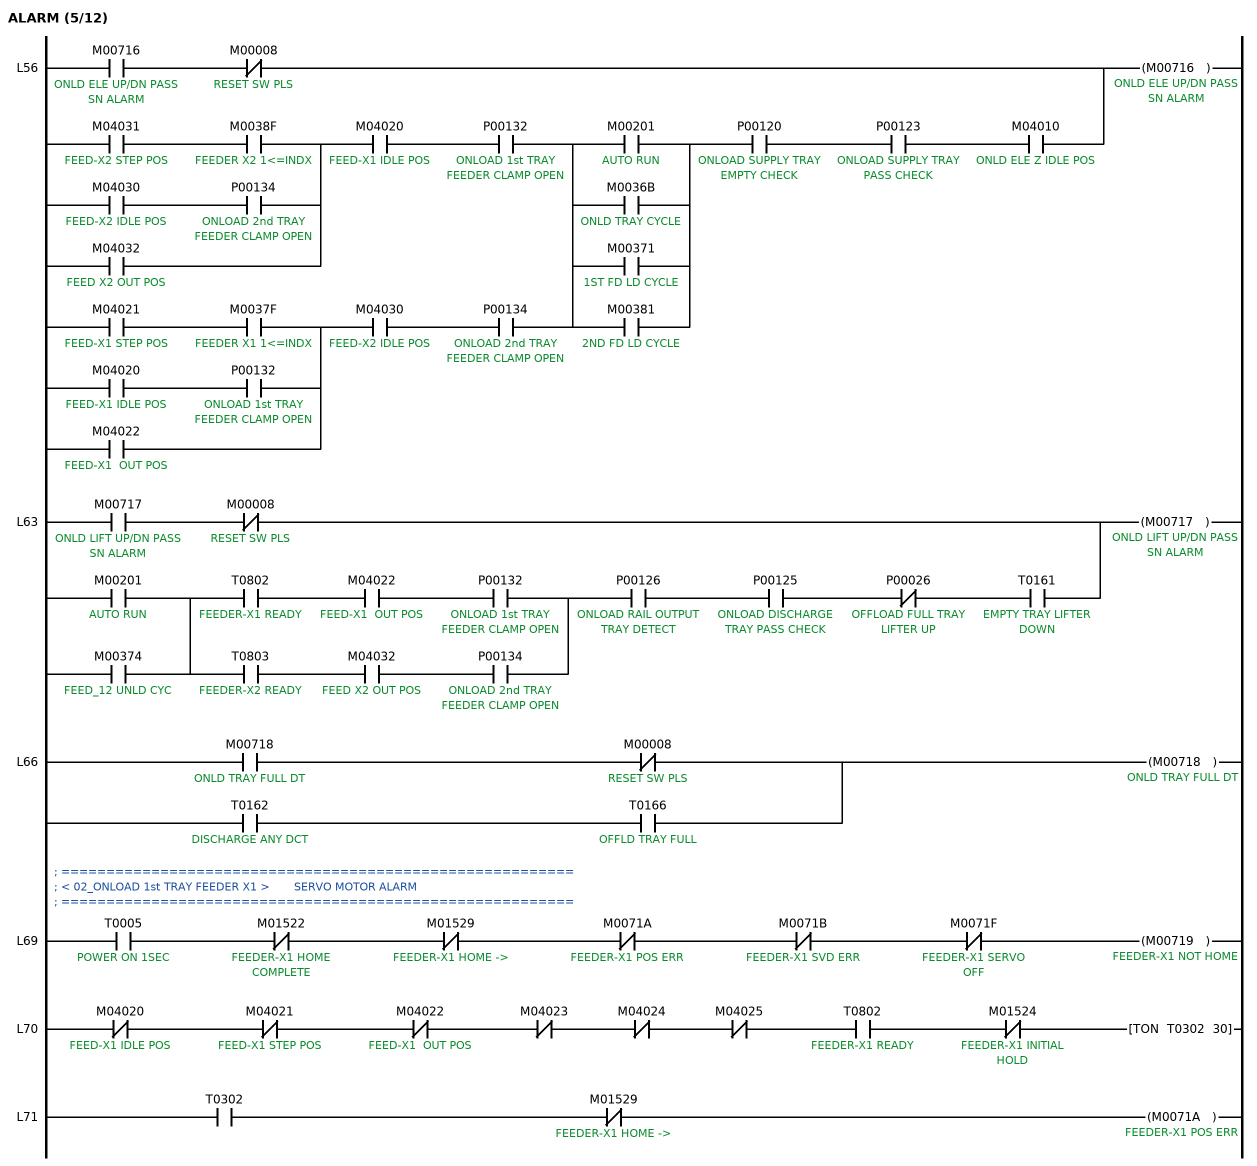
; L56
LOAD      M00716	// ONLD ELE UP/DN PASS SN ALARM
AND NOT   M00008	// RESET SW PLS
LOAD      M04031	// FEED-X2 STEP POS
AND       M0038F	// FEEDER X2 1<=INDX
LOAD      M04030	// FEED-X2 IDLE POS
AND       P00134	// ONLOAD 2nd TRAY FEEDER CLAMP OPEN
OR LOAD
OR        M04032	// FEED X2 OUT POS
AND       M04020	// FEED-X1 IDLE POS
AND       P00132	// ONLOAD 1st TRAY FEEDER CLAMP OPEN
LOAD      M04021	// FEED-X1 STEP POS
AND       M0037F	// FEEDER X1 1<=INDX
LOAD      M04020	// FEED-X1 IDLE POS
AND       P00132	// ONLOAD 1st TRAY FEEDER CLAMP OPEN
OR LOAD
OR        M04022	// FEED-X1  OUT POS
AND       M04030	// FEED-X2 IDLE POS
AND       P00134	// ONLOAD 2nd TRAY FEEDER CLAMP OPEN
OR LOAD
LOAD      M00201	// AUTO RUN
OR        M0036B	// ONLD TRAY CYCLE
OR        M00371	// 1ST FD LD CYCLE
OR        M00381	// 2ND FD LD CYCLE
AND LOAD
AND       P00120	// ONLOAD SUPPLY TRAY EMPTY CHECK
AND       P00123	// ONLOAD SUPPLY TRAY PASS CHECK
AND       M04010	// ONLD ELE Z IDLE POS
OR LOAD
OUT       M00716	// ONLD ELE UP/DN PASS SN ALARM
; L63
LOAD      M00717	// ONLD LIFT UP/DN PASS SN ALARM
AND NOT   M00008	// RESET SW PLS
LOAD      M00201	// AUTO RUN
OR        M00374	// FEED_12 UNLD CYC
LOAD      T0802	// FEEDER-X1 READY
AND       M04022	// FEED-X1  OUT POS
AND       P00132	// ONLOAD 1st TRAY FEEDER CLAMP OPEN
LOAD      T0803	// FEEDER-X2 READY
AND       M04032	// FEED X2 OUT POS
AND       P00134	// ONLOAD 2nd TRAY FEEDER CLAMP OPEN
OR LOAD
AND LOAD
AND       P00126	// ONLOAD RAIL OUTPUT TRAY DETECT
AND       P00125	// ONLOAD DISCHARGE TRAY PASS CHECK
AND NOT   P00026	// OFFLOAD FULL TRAY LIFTER UP
AND       T0161	// EMPTY TRAY LIFTER DOWN
OR LOAD
OUT       M00717	// ONLD LIFT UP/DN PASS SN ALARM
; L66
LOAD      M00718	// ONLD TRAY FULL DT
AND NOT   M00008	// RESET SW PLS
LOAD      T0162	// DISCHARGE ANY DCT
AND       T0166	// OFFLD TRAY FULL
OR LOAD
OUT       M00718	// ONLD TRAY FULL DT
// =========================================================
// 
//        < 02_ONLOAD 1st TRAY FEEDER X1 >       SERVO MOTOR ALARM
// 
// =========================================================
; L69
LOAD      T0005	// POWER ON 1SEC
AND NOT   M01522	// FEEDER-X1 HOME COMPLETE
AND NOT   M01529	// FEEDER-X1 HOME ->
AND NOT   M0071A	// FEEDER-X1 POS ERR
AND NOT   M0071B	// FEEDER-X1 SVD ERR
AND NOT   M0071F	// FEEDER-X1 SERVO OFF
OUT       M00719	// FEEDER-X1 NOT HOME
; L70
LOAD NOT  M04020	// FEED-X1 IDLE POS
AND NOT   M04021	// FEED-X1 STEP POS
AND NOT   M04022	// FEED-X1  OUT POS
AND NOT   M04023
AND NOT   M04024
AND NOT   M04025
AND       T0802	// FEEDER-X1 READY
AND NOT   M01524	// FEEDER-X1 INITIAL HOLD
TON       T0302 30
; L71
LOAD      T0302
AND NOT   M01529	// FEEDER-X1 HOME ->
OUT       M0071A	// FEEDER-X1 POS ERR

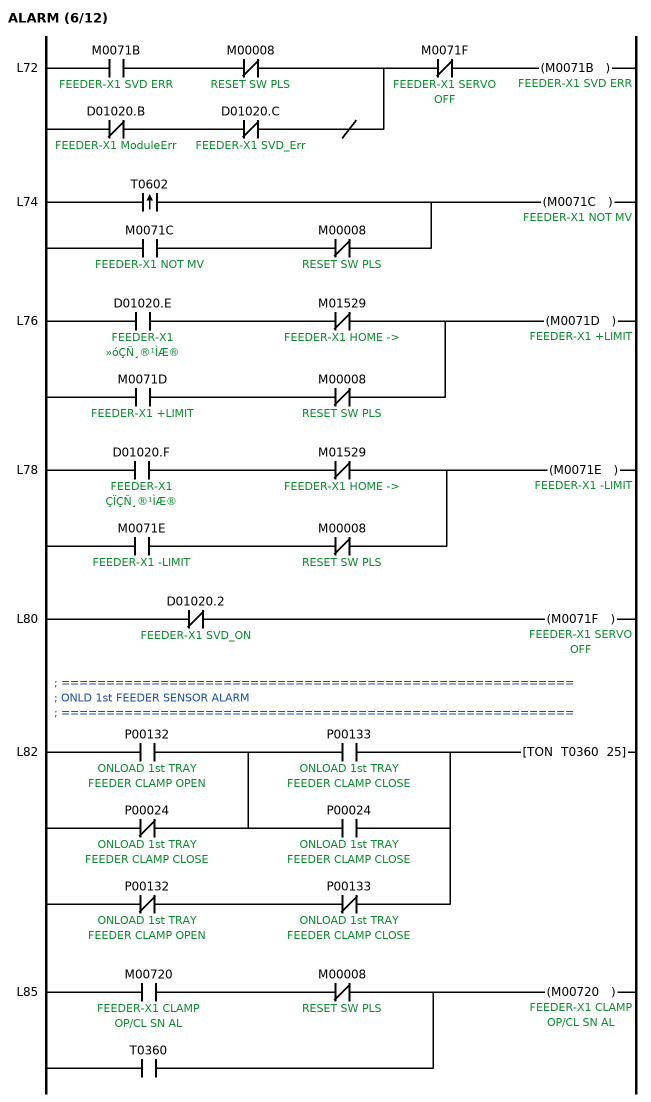
; L72
LOAD      M0071B	// FEEDER-X1 SVD ERR
AND NOT   M00008	// RESET SW PLS
LOAD NOT  D01020.B	// FEEDER-X1 ModuleErr
AND NOT   D01020.C	// FEEDER-X1 SVD_Err
NOT
OR LOAD
AND NOT   M0071F	// FEEDER-X1 SERVO OFF
OUT       M0071B	// FEEDER-X1 SVD ERR
; L74
LOADP     T0602
LOAD      M0071C	// FEEDER-X1 NOT MV
AND NOT   M00008	// RESET SW PLS
OR LOAD
OUT       M0071C	// FEEDER-X1 NOT MV
; L76
LOAD      D01020.E	// FEEDER-X1 »óÇÑ¸®¹ÌÆ®
AND NOT   M01529	// FEEDER-X1 HOME ->
LOAD      M0071D	// FEEDER-X1 +LIMIT
AND NOT   M00008	// RESET SW PLS
OR LOAD
OUT       M0071D	// FEEDER-X1 +LIMIT
; L78
LOAD      D01020.F	// FEEDER-X1 ÇÏÇÑ¸®¹ÌÆ®
AND NOT   M01529	// FEEDER-X1 HOME ->
LOAD      M0071E	// FEEDER-X1 -LIMIT
AND NOT   M00008	// RESET SW PLS
OR LOAD
OUT       M0071E	// FEEDER-X1 -LIMIT
; L80
LOAD NOT  D01020.2	// FEEDER-X1 SVD_ON
OUT       M0071F	// FEEDER-X1 SERVO OFF
// =========================================================
// 
//        ONLD 1st FEEDER SENSOR ALARM
// 
// =========================================================
; L82
LOAD      P00132	// ONLOAD 1st TRAY FEEDER CLAMP OPEN
OR NOT    P00024	// ONLOAD 1st TRAY FEEDER CLAMP CLOSE
LOAD      P00133	// ONLOAD 1st TRAY FEEDER CLAMP CLOSE
OR        P00024	// ONLOAD 1st TRAY FEEDER CLAMP CLOSE
AND LOAD
LOAD NOT  P00132	// ONLOAD 1st TRAY FEEDER CLAMP OPEN
AND NOT   P00133	// ONLOAD 1st TRAY FEEDER CLAMP CLOSE
OR LOAD
TON       T0360 25
; L85
LOAD      M00720	// FEEDER-X1 CLAMP OP/CL SN AL
AND NOT   M00008	// RESET SW PLS
OR        T0360
OUT       M00720	// FEEDER-X1 CLAMP OP/CL SN AL

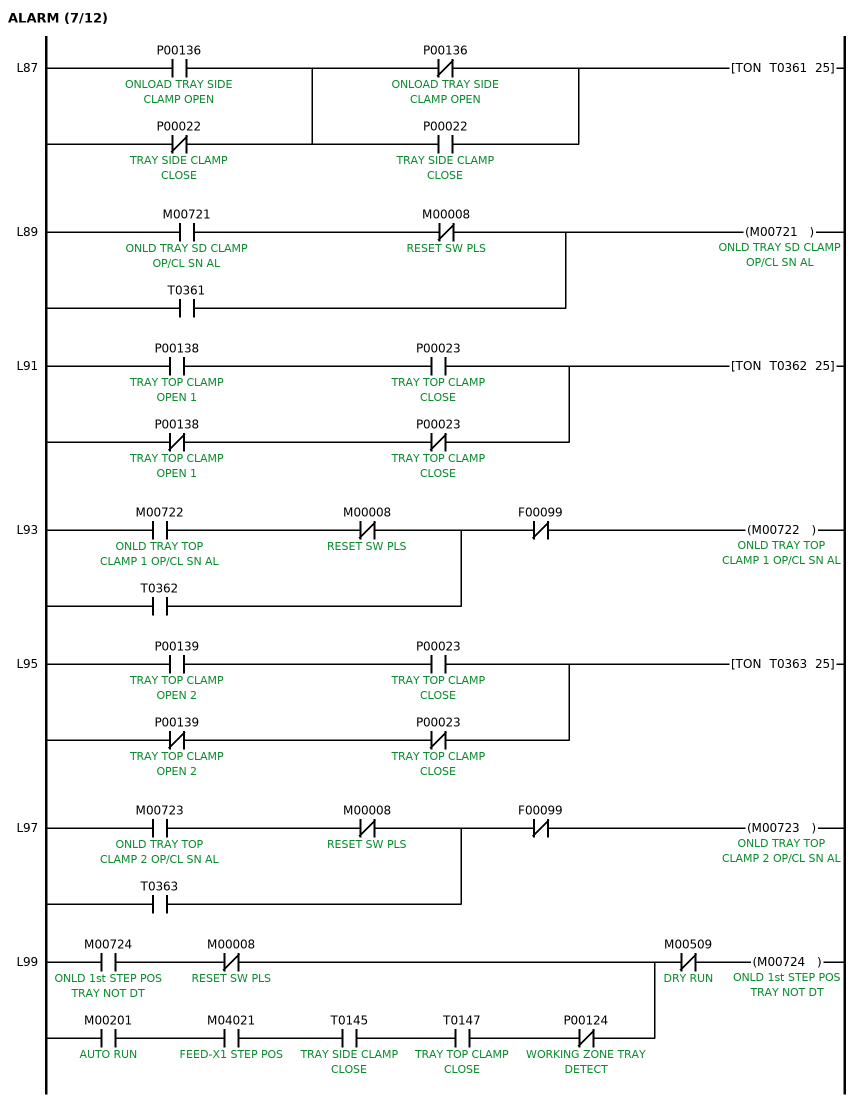
; L87
LOAD      P00136	// ONLOAD TRAY SIDE CLAMP OPEN
OR NOT    P00022	// TRAY SIDE CLAMP CLOSE
LOAD NOT  P00136	// ONLOAD TRAY SIDE CLAMP OPEN
OR        P00022	// TRAY SIDE CLAMP CLOSE
AND LOAD
TON       T0361 25
; L89
LOAD      M00721	// ONLD TRAY SD CLAMP OP/CL SN AL
AND NOT   M00008	// RESET SW PLS
OR        T0361
OUT       M00721	// ONLD TRAY SD CLAMP OP/CL SN AL
; L91
LOAD      P00138	// TRAY TOP CLAMP OPEN 1
AND       P00023	// TRAY TOP CLAMP CLOSE
LOAD NOT  P00138	// TRAY TOP CLAMP OPEN 1
AND NOT   P00023	// TRAY TOP CLAMP CLOSE
OR LOAD
TON       T0362 25
; L93
LOAD      M00722	// ONLD TRAY TOP CLAMP 1 OP/CL SN AL
AND NOT   M00008	// RESET SW PLS
OR        T0362
AND NOT   F00099
OUT       M00722	// ONLD TRAY TOP CLAMP 1 OP/CL SN AL
; L95
LOAD      P00139	// TRAY TOP CLAMP OPEN 2
AND       P00023	// TRAY TOP CLAMP CLOSE
LOAD NOT  P00139	// TRAY TOP CLAMP OPEN 2
AND NOT   P00023	// TRAY TOP CLAMP CLOSE
OR LOAD
TON       T0363 25
; L97
LOAD      M00723	// ONLD TRAY TOP CLAMP 2 OP/CL SN AL
AND NOT   M00008	// RESET SW PLS
OR        T0363
AND NOT   F00099
OUT       M00723	// ONLD TRAY TOP CLAMP 2 OP/CL SN AL
; L99
LOAD      M00724	// ONLD 1st STEP POS TRAY NOT DT
AND NOT   M00008	// RESET SW PLS
LOAD      M00201	// AUTO RUN
AND       M04021	// FEED-X1 STEP POS
AND       T0145	// TRAY SIDE CLAMP CLOSE
AND       T0147	// TRAY TOP CLAMP CLOSE
AND NOT   P00124	// WORKING ZONE TRAY DETECT
OR LOAD
AND NOT   M00509	// DRY RUN
OUT       M00724	// ONLD 1st STEP POS TRAY NOT DT

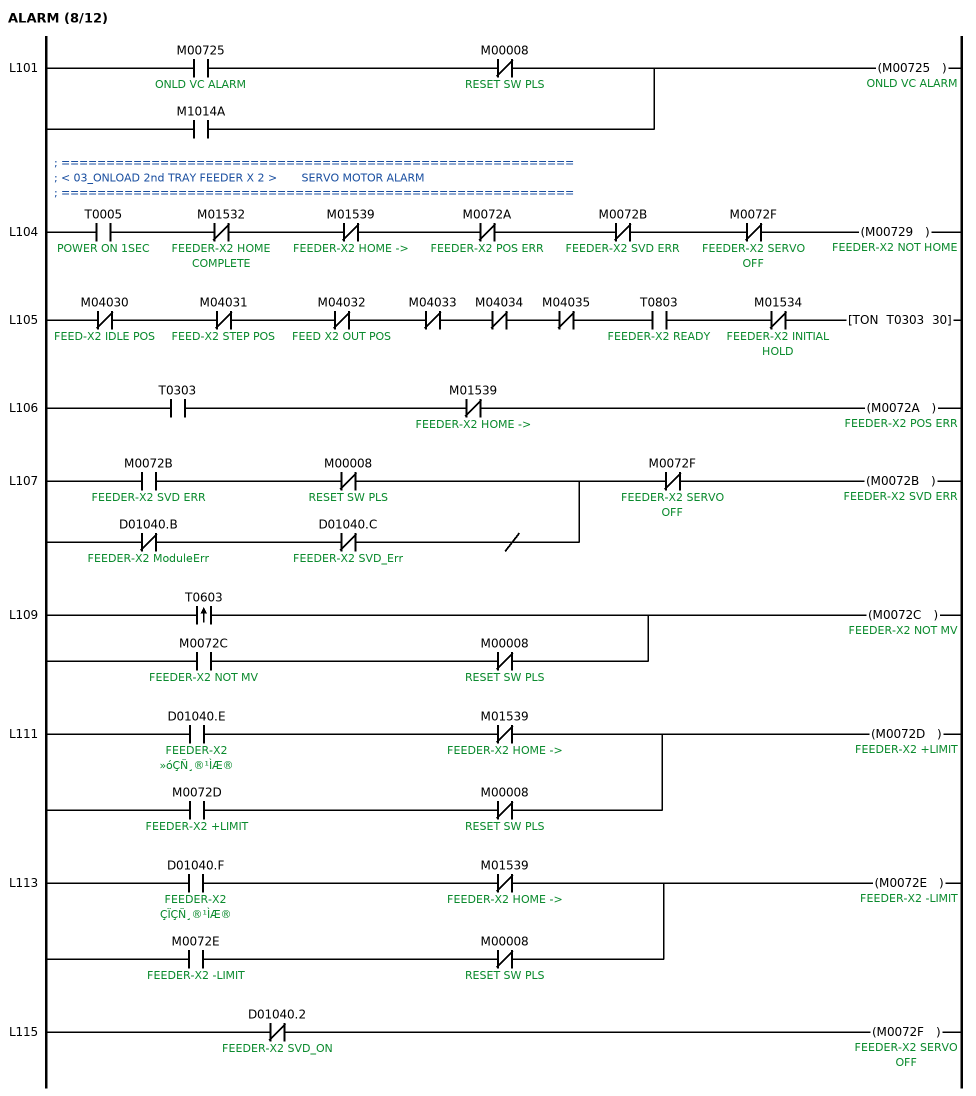
; L101
LOAD      M00725	// ONLD VC ALARM
AND NOT   M00008	// RESET SW PLS
OR        M1014A
OUT       M00725	// ONLD VC ALARM
// =========================================================
// 
//        < 03_ONLOAD 2nd TRAY FEEDER X 2 >       SERVO MOTOR ALARM
// 
// =========================================================
; L104
LOAD      T0005	// POWER ON 1SEC
AND NOT   M01532	// FEEDER-X2 HOME COMPLETE
AND NOT   M01539	// FEEDER-X2 HOME ->
AND NOT   M0072A	// FEEDER-X2 POS ERR
AND NOT   M0072B	// FEEDER-X2 SVD ERR
AND NOT   M0072F	// FEEDER-X2 SERVO OFF
OUT       M00729	// FEEDER-X2 NOT HOME
; L105
LOAD NOT  M04030	// FEED-X2 IDLE POS
AND NOT   M04031	// FEED-X2 STEP POS
AND NOT   M04032	// FEED X2 OUT POS
AND NOT   M04033
AND NOT   M04034
AND NOT   M04035
AND       T0803	// FEEDER-X2 READY
AND NOT   M01534	// FEEDER-X2 INITIAL HOLD
TON       T0303 30
; L106
LOAD      T0303
AND NOT   M01539	// FEEDER-X2 HOME ->
OUT       M0072A	// FEEDER-X2 POS ERR
; L107
LOAD      M0072B	// FEEDER-X2 SVD ERR
AND NOT   M00008	// RESET SW PLS
LOAD NOT  D01040.B	// FEEDER-X2 ModuleErr
AND NOT   D01040.C	// FEEDER-X2 SVD_Err
NOT
OR LOAD
AND NOT   M0072F	// FEEDER-X2 SERVO OFF
OUT       M0072B	// FEEDER-X2 SVD ERR
; L109
LOADP     T0603
LOAD      M0072C	// FEEDER-X2 NOT MV
AND NOT   M00008	// RESET SW PLS
OR LOAD
OUT       M0072C	// FEEDER-X2 NOT MV
; L111
LOAD      D01040.E	// FEEDER-X2 »óÇÑ¸®¹ÌÆ®
AND NOT   M01539	// FEEDER-X2 HOME ->
LOAD      M0072D	// FEEDER-X2 +LIMIT
AND NOT   M00008	// RESET SW PLS
OR LOAD
OUT       M0072D	// FEEDER-X2 +LIMIT
; L113
LOAD      D01040.F	// FEEDER-X2 ÇÏÇÑ¸®¹ÌÆ®
AND NOT   M01539	// FEEDER-X2 HOME ->
LOAD      M0072E	// FEEDER-X2 -LIMIT
AND NOT   M00008	// RESET SW PLS
OR LOAD
OUT       M0072E	// FEEDER-X2 -LIMIT
; L115
LOAD NOT  D01040.2	// FEEDER-X2 SVD_ON
OUT       M0072F	// FEEDER-X2 SERVO OFF

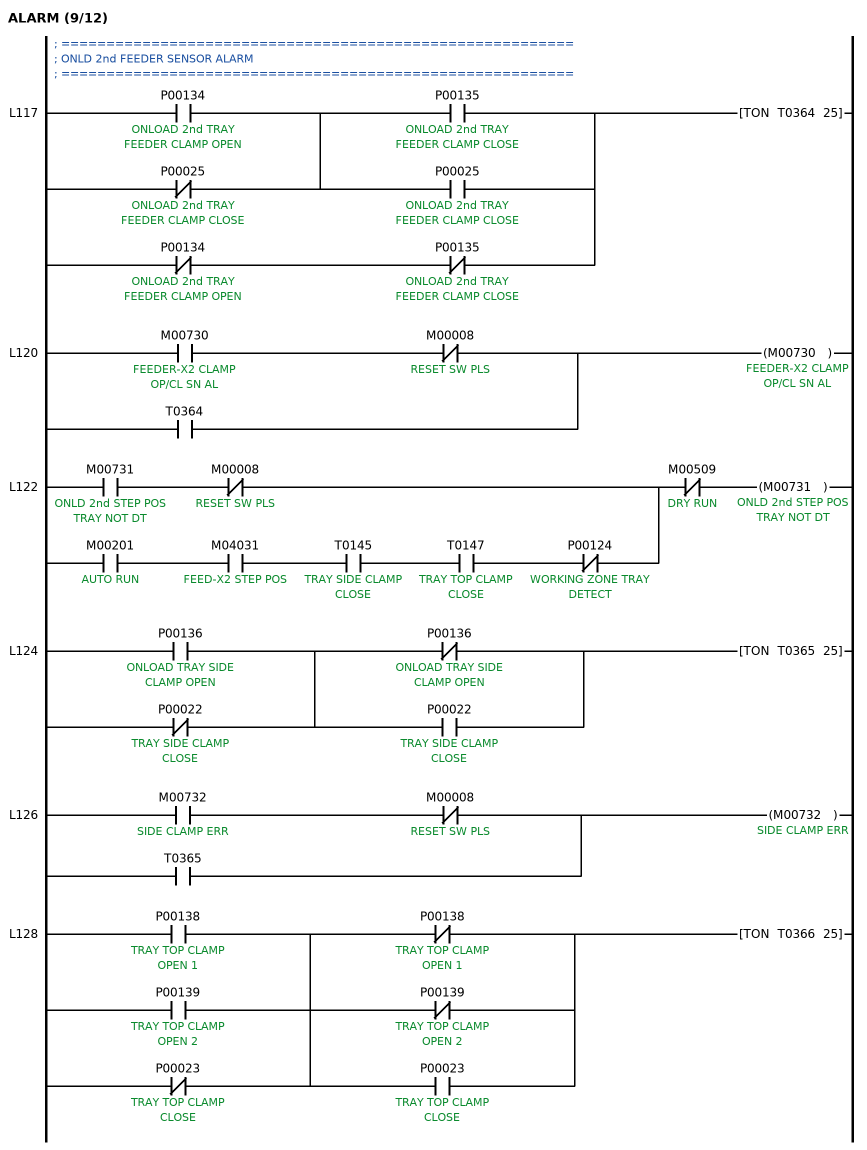
// =========================================================
// 
//        ONLD 2nd FEEDER SENSOR ALARM
// 
// =========================================================
; L117
LOAD      P00134	// ONLOAD 2nd TRAY FEEDER CLAMP OPEN
OR NOT    P00025	// ONLOAD 2nd TRAY FEEDER CLAMP CLOSE
LOAD      P00135	// ONLOAD 2nd TRAY FEEDER CLAMP CLOSE
OR        P00025	// ONLOAD 2nd TRAY FEEDER CLAMP CLOSE
AND LOAD
LOAD NOT  P00134	// ONLOAD 2nd TRAY FEEDER CLAMP OPEN
AND NOT   P00135	// ONLOAD 2nd TRAY FEEDER CLAMP CLOSE
OR LOAD
TON       T0364 25
; L120
LOAD      M00730	// FEEDER-X2 CLAMP OP/CL SN AL
AND NOT   M00008	// RESET SW PLS
OR        T0364
OUT       M00730	// FEEDER-X2 CLAMP OP/CL SN AL
; L122
LOAD      M00731	// ONLD 2nd STEP POS TRAY NOT DT
AND NOT   M00008	// RESET SW PLS
LOAD      M00201	// AUTO RUN
AND       M04031	// FEED-X2 STEP POS
AND       T0145	// TRAY SIDE CLAMP CLOSE
AND       T0147	// TRAY TOP CLAMP CLOSE
AND NOT   P00124	// WORKING ZONE TRAY DETECT
OR LOAD
AND NOT   M00509	// DRY RUN
OUT       M00731	// ONLD 2nd STEP POS TRAY NOT DT
; L124
LOAD      P00136	// ONLOAD TRAY SIDE CLAMP OPEN
OR NOT    P00022	// TRAY SIDE CLAMP CLOSE
LOAD NOT  P00136	// ONLOAD TRAY SIDE CLAMP OPEN
OR        P00022	// TRAY SIDE CLAMP CLOSE
AND LOAD
TON       T0365 25
; L126
LOAD      M00732	// SIDE CLAMP ERR
AND NOT   M00008	// RESET SW PLS
OR        T0365
OUT       M00732	// SIDE CLAMP ERR
; L128
LOAD      P00138	// TRAY TOP CLAMP OPEN 1
OR        P00139	// TRAY TOP CLAMP OPEN 2
OR NOT    P00023	// TRAY TOP CLAMP CLOSE
LOAD NOT  P00138	// TRAY TOP CLAMP OPEN 1
OR NOT    P00139	// TRAY TOP CLAMP OPEN 2
OR        P00023	// TRAY TOP CLAMP CLOSE
AND LOAD
TON       T0366 25

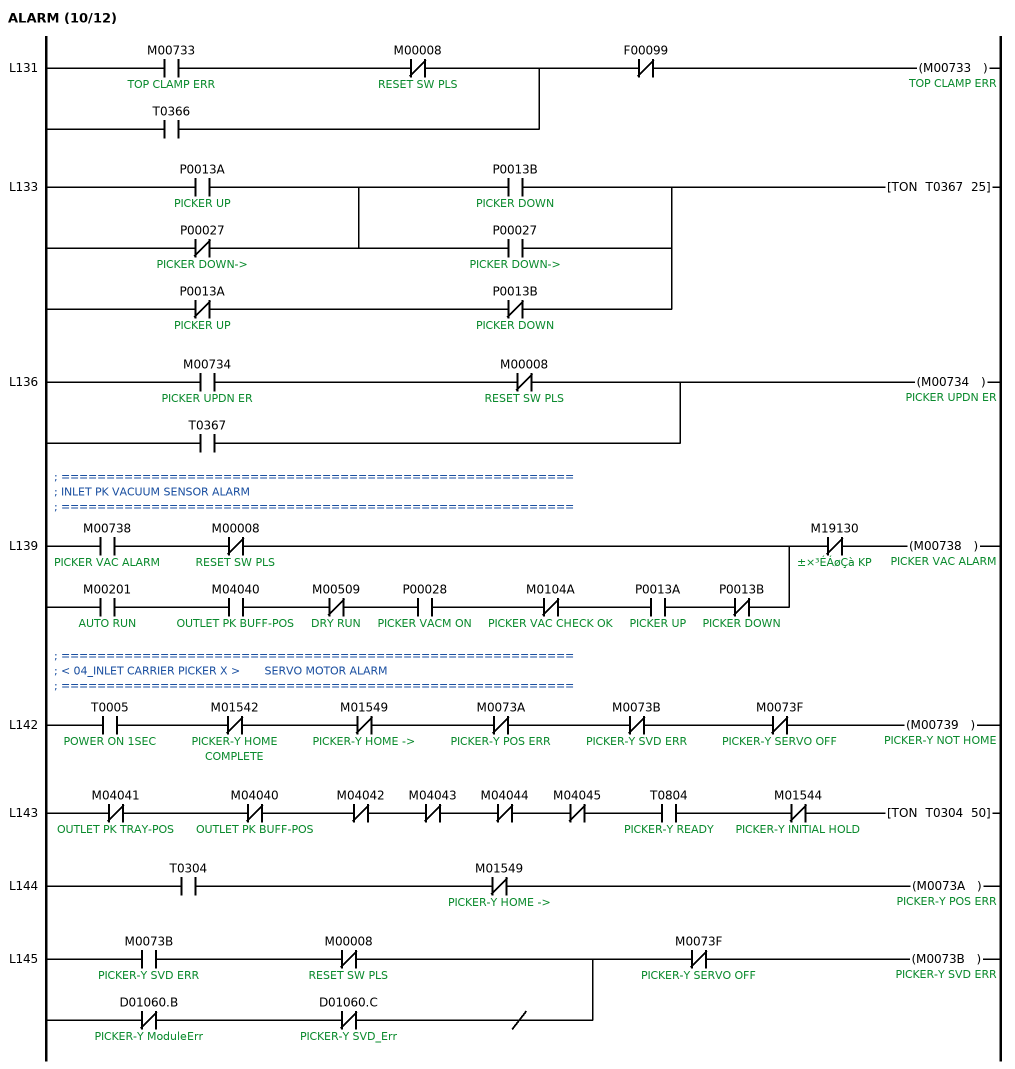
; L131
LOAD      M00733	// TOP CLAMP ERR
AND NOT   M00008	// RESET SW PLS
OR        T0366
AND NOT   F00099
OUT       M00733	// TOP CLAMP ERR
; L133
LOAD      P0013A	// PICKER UP
OR NOT    P00027	// PICKER DOWN->
LOAD      P0013B	// PICKER DOWN
OR        P00027	// PICKER DOWN->
AND LOAD
LOAD NOT  P0013A	// PICKER UP
AND NOT   P0013B	// PICKER DOWN
OR LOAD
TON       T0367 25
; L136
LOAD      M00734	// PICKER UPDN ER
AND NOT   M00008	// RESET SW PLS
OR        T0367
OUT       M00734	// PICKER UPDN ER
// =========================================================
// 
//        INLET PK VACUUM SENSOR ALARM
// 
// =========================================================
; L139
LOAD      M00738	// PICKER VAC ALARM
AND NOT   M00008	// RESET SW PLS
LOAD      M00201	// AUTO RUN
AND       M04040	// OUTLET PK BUFF-POS
AND NOT   M00509	// DRY RUN
AND       P00028	// PICKER VACM ON
AND NOT   M0104A	// PICKER VAC CHECK OK
AND       P0013A	// PICKER UP
AND NOT   P0013B	// PICKER DOWN
OR LOAD
AND NOT   M19130	// ±×³ÉÁøÇà KP
OUT       M00738	// PICKER VAC ALARM
// =========================================================
// 
//        < 04_INLET CARRIER PICKER X >       SERVO MOTOR ALARM
// 
// =========================================================
; L142
LOAD      T0005	// POWER ON 1SEC
AND NOT   M01542	// PICKER-Y HOME COMPLETE
AND NOT   M01549	// PICKER-Y HOME ->
AND NOT   M0073A	// PICKER-Y POS ERR
AND NOT   M0073B	// PICKER-Y SVD ERR
AND NOT   M0073F	// PICKER-Y SERVO OFF
OUT       M00739	// PICKER-Y NOT HOME
; L143
LOAD NOT  M04041	// OUTLET PK TRAY-POS
AND NOT   M04040	// OUTLET PK BUFF-POS
AND NOT   M04042
AND NOT   M04043
AND NOT   M04044
AND NOT   M04045
AND       T0804	// PICKER-Y READY
AND NOT   M01544	// PICKER-Y INITIAL HOLD
TON       T0304 50
; L144
LOAD      T0304
AND NOT   M01549	// PICKER-Y HOME ->
OUT       M0073A	// PICKER-Y POS ERR
; L145
LOAD      M0073B	// PICKER-Y SVD ERR
AND NOT   M00008	// RESET SW PLS
LOAD NOT  D01060.B	// PICKER-Y ModuleErr
AND NOT   D01060.C	// PICKER-Y SVD_Err
NOT
OR LOAD
AND NOT   M0073F	// PICKER-Y SERVO OFF
OUT       M0073B	// PICKER-Y SVD ERR

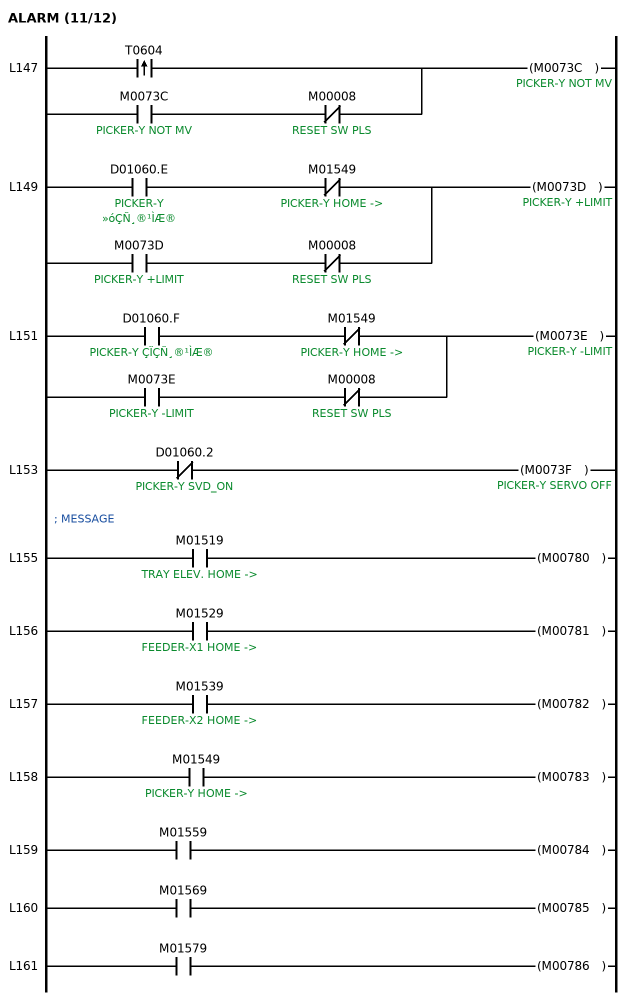
; L147
LOADP     T0604
LOAD      M0073C	// PICKER-Y NOT MV
AND NOT   M00008	// RESET SW PLS
OR LOAD
OUT       M0073C	// PICKER-Y NOT MV
; L149
LOAD      D01060.E	// PICKER-Y »óÇÑ¸®¹ÌÆ®
AND NOT   M01549	// PICKER-Y HOME ->
LOAD      M0073D	// PICKER-Y +LIMIT
AND NOT   M00008	// RESET SW PLS
OR LOAD
OUT       M0073D	// PICKER-Y +LIMIT
; L151
LOAD      D01060.F	// PICKER-Y ÇÏÇÑ¸®¹ÌÆ®
AND NOT   M01549	// PICKER-Y HOME ->
LOAD      M0073E	// PICKER-Y -LIMIT
AND NOT   M00008	// RESET SW PLS
OR LOAD
OUT       M0073E	// PICKER-Y -LIMIT
; L153
LOAD NOT  D01060.2	// PICKER-Y SVD_ON
OUT       M0073F	// PICKER-Y SERVO OFF
// MESSAGE
; L155
LOAD      M01519	// TRAY ELEV. HOME ->
OUT       M00780
; L156
LOAD      M01529	// FEEDER-X1 HOME ->
OUT       M00781
; L157
LOAD      M01539	// FEEDER-X2 HOME ->
OUT       M00782
; L158
LOAD      M01549	// PICKER-Y HOME ->
OUT       M00783
; L159
LOAD      M01559
OUT       M00784
; L160
LOAD      M01569
OUT       M00785
; L161
LOAD      M01579
OUT       M00786

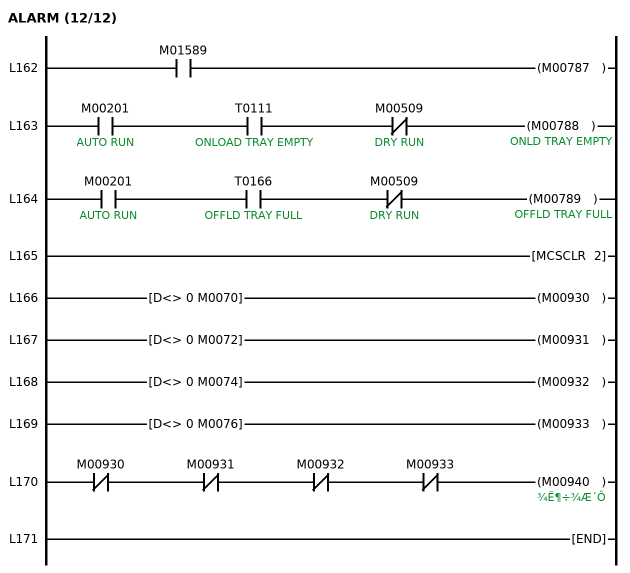
; L162
LOAD      M01589
OUT       M00787
; L163
LOAD      M00201	// AUTO RUN
AND       T0111	// ONLOAD TRAY EMPTY
AND NOT   M00509	// DRY RUN
OUT       M00788	// ONLD TRAY EMPTY
; L164
LOAD      M00201	// AUTO RUN
AND       T0166	// OFFLD TRAY FULL
AND NOT   M00509	// DRY RUN
OUT       M00789	// OFFLD TRAY FULL
; L165
MCSCLR    2
; L166
LOADD<>   0 M0070
OUT       M00930
; L167
LOADD<>   0 M0072
OUT       M00931
; L168
LOADD<>   0 M0074
OUT       M00932
; L169
LOADD<>   0 M0076
OUT       M00933
; L170
LOAD NOT  M00930
AND NOT   M00931
AND NOT   M00932
AND NOT   M00933
OUT       M00940	// ¾Ë¶÷¾Æ´Ô
; L171
END

PROGRAM DEVICE_CHANGE (task: ½ºÄµ ÇÁ·Î±×·¥)

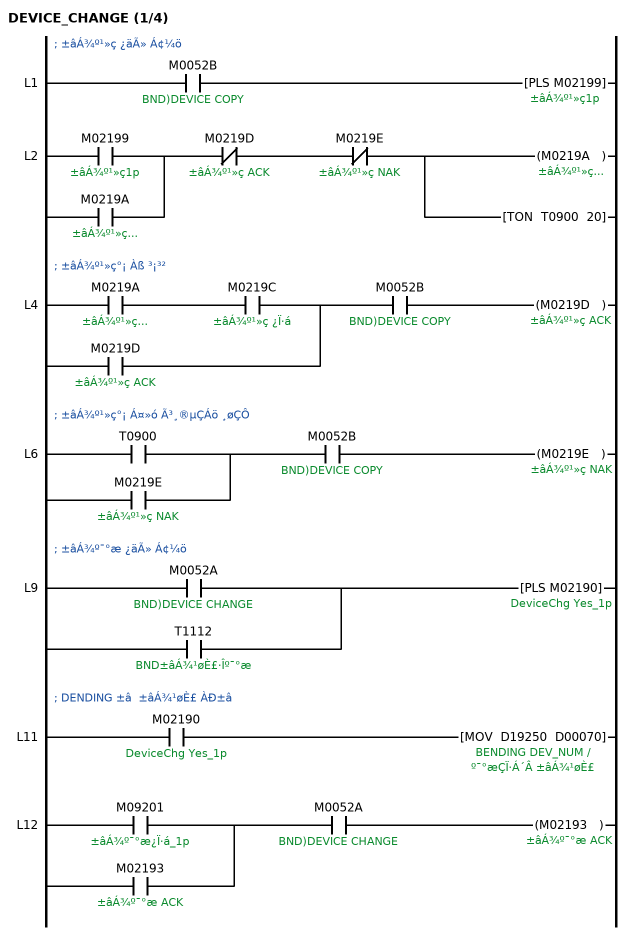
// ±âÁ¾º¹»ç ¿äÃ» Á¢¼ö
; L1
LOAD      M0052B	// BND)DEVICE COPY
OUTP      M02199	// ±âÁ¾º¹»ç1p
; L2
LOAD      M02199	// ±âÁ¾º¹»ç1p
OR        M0219A	// ±âÁ¾º¹»ç...
AND NOT   M0219D	// ±âÁ¾º¹»ç ACK
AND NOT   M0219E	// ±âÁ¾º¹»ç NAK
OUT       M0219A	// ±âÁ¾º¹»ç...
TON       T0900 20
; L4
LOAD      M0219A	// ±âÁ¾º¹»ç...
AND       M0219C	// ±âÁ¾º¹»ç ¿Ï·á
OR        M0219D	// ±âÁ¾º¹»ç ACK
AND       M0052B	// BND)DEVICE COPY
OUT       M0219D	// ±âÁ¾º¹»ç ACK
// output comment: ±âÁ¾º¹»ç°¡ Àß ³¡³²
; L6
LOAD      T0900
OR        M0219E	// ±âÁ¾º¹»ç NAK
AND       M0052B	// BND)DEVICE COPY
OUT       M0219E	// ±âÁ¾º¹»ç NAK
// output comment: ±âÁ¾º¹»ç°¡ Á¤»ó Ã³¸®µÇÁö ¸øÇÔ
// ±âÁ¾º¯°æ ¿äÃ» Á¢¼ö
; L9
LOAD      M0052A	// BND)DEVICE CHANGE
OR        T1112	// BND±âÁ¾¹øÈ£·Îº¯°æ
OUTP      M02190	// DeviceChg Yes_1p
; L11
LOAD      M02190	// DeviceChg Yes_1p
MOV       D19250 D00070	// BENDING DEV_NUM / º¯°æÇÏ·Á´Â ±âÁ¾¹øÈ£
// output comment: DENDING ±â  ±âÁ¾¹øÈ£ ÀÐ±â
; L12
LOAD      M09201	// ±âÁ¾º¯°æ¿Ï·á_1p
OR        M02193	// ±âÁ¾º¯°æ ACK
AND       M0052A	// BND)DEVICE CHANGE
OUT       M02193	// ±âÁ¾º¯°æ ACK

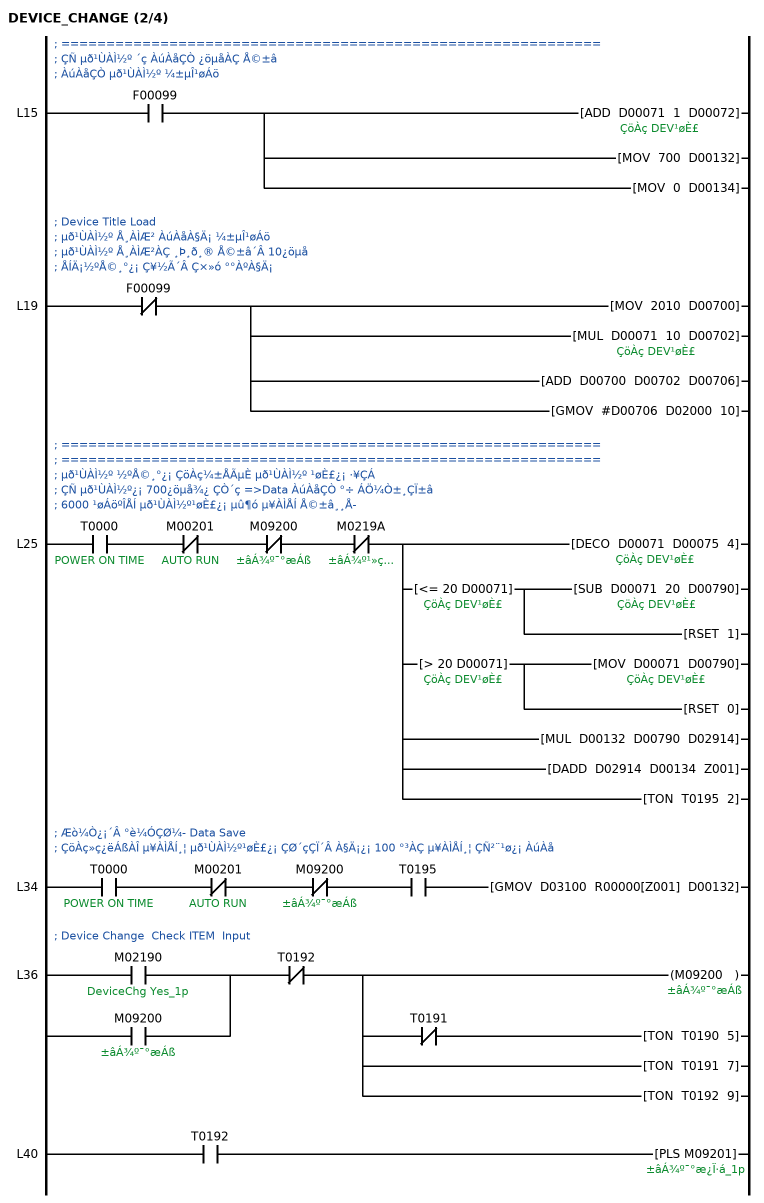
// ============================================================
; L15
LOAD      F00099
ADD       D00071 1 D00072	// ÇöÀç DEV¹øÈ£
MOV       700 D00132
MOV       0 D00134
// output comment: ÇÑ µð¹ÙÀÌ½º ´ç ÀúÀåÇÒ ¿öµåÀÇ Å©±â
// output comment: ÀúÀåÇÒ µð¹ÙÀÌ½º ¼±µÎ¹øÁö
// Device Title Load
; L19
LOAD NOT  F00099
MOV       2010 D00700
MUL       D00071 10 D00702	// ÇöÀç DEV¹øÈ£
ADD       D00700 D00702 D00706
GMOV      #D00706 D02000 10
// output comment: µð¹ÙÀÌ½º Å¸ÀÌÆ² ÀúÀåÀ§Ä¡ ¼±µÎ¹øÁö
// output comment: µð¹ÙÀÌ½º Å¸ÀÌÆ²ÀÇ ¸Þ¸ð¸® Å©±â´Â 10¿öµå
// output comment: ÅÍÄ¡½ºÅ©¸°¿¡ Ç¥½Ã´Â Ç×»ó °°ÀºÀ§Ä¡
// ============================================================
// ============================================================
; L25
LOAD      T0000	// POWER ON TIME
AND NOT   M00201	// AUTO RUN
AND NOT   M09200	// ±âÁ¾º¯°æÁß
AND NOT   M0219A	// ±âÁ¾º¹»ç...
DECO      D00071 D00075 4	// ÇöÀç DEV¹øÈ£
MPUSH
AND<=     20 D00071	// ÇöÀç DEV¹øÈ£
SUB       D00071 20 D00790	// ÇöÀç DEV¹øÈ£
RSET      1
MLOAD
AND>      20 D00071	// ÇöÀç DEV¹øÈ£
MOV       D00071 D00790	// ÇöÀç DEV¹øÈ£
RSET      0
MPOP
MUL       D00132 D00790 D02914
DADD      D02914 D00134 Z001
TON       T0195 2
// output comment: µð¹ÙÀÌ½º ½ºÅ©¸°¿¡ ÇöÀç¼±ÅÃµÈ µð¹ÙÀÌ½º ¹øÈ£¿¡ ·¥ÇÁ
// output comment: ÇÑ µð¹ÙÀÌ½º¿¡ 700¿öµå¾¿ ÇÒ´ç =>Data ÀúÀåÇÒ °÷ ÁÖ¼Ò±¸ÇÏ±â
// output comment: 6000 ¹øÁöºÎÅÍ µð¹ÙÀÌ½º¹øÈ£¿¡ µû¶ó µ¥ÀÌÅÍ Å©±â¸¸Å­
// Æò¼Ò¿¡´Â °è¼ÓÇØ¼­ Data Save
; L34
LOAD      T0000	// POWER ON TIME
AND NOT   M00201	// AUTO RUN
AND NOT   M09200	// ±âÁ¾º¯°æÁß
AND       T0195
GMOV      D03100 R00000[Z001] D00132
// output comment: ÇöÀç»ç¿ëÁßÀÎ µ¥ÀÌÅÍ¸¦ µð¹ÙÀÌ½º¹øÈ£¿¡ ÇØ´çÇÏ´Â À§Ä¡¿¡ 100 °³ÀÇ µ¥ÀÌÅÍ¸¦ ÇÑ²¨¹ø¿¡ ÀúÀå
// Device Change  Check ITEM  Input
; L36
LOAD      M02190	// DeviceChg Yes_1p
OR        M09200	// ±âÁ¾º¯°æÁß
AND NOT   T0192
OUT       M09200	// ±âÁ¾º¯°æÁß
MPUSH
AND NOT   T0191
TON       T0190 5
MPOP
TON       T0191 7
TON       T0192 9
; L40
LOAD      T0192
OUTP      M09201	// ±âÁ¾º¯°æ¿Ï·á_1p

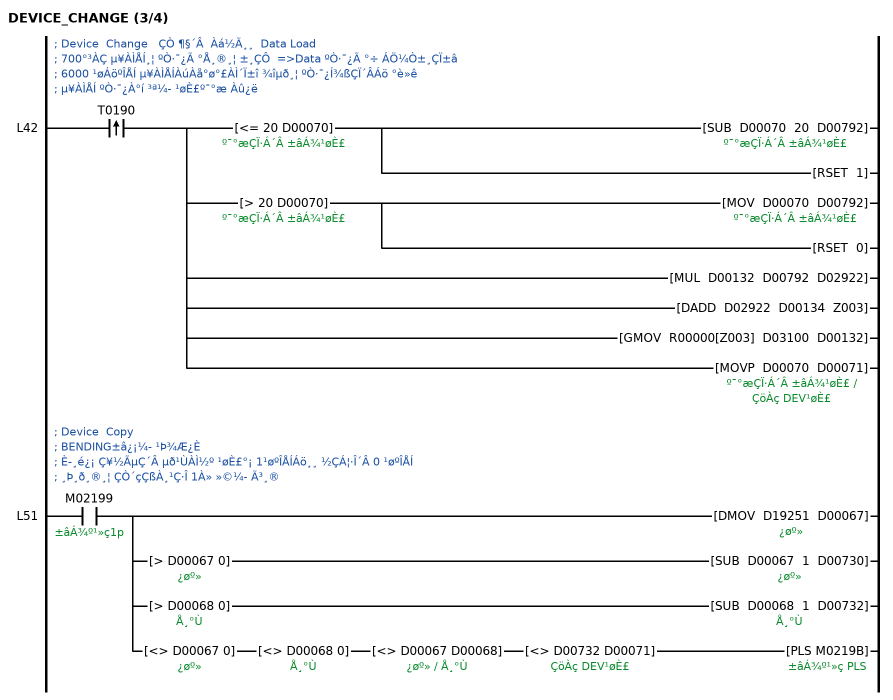
// Device  Change   ÇÒ ¶§´Â  Àá½Ã¸¸  Data Load
; L42
LOADP     T0190
MPUSH
AND<=     20 D00070	// º¯°æÇÏ·Á´Â ±âÁ¾¹øÈ£
SUB       D00070 20 D00792	// º¯°æÇÏ·Á´Â ±âÁ¾¹øÈ£
RSET      1
MLOAD
AND>      20 D00070	// º¯°æÇÏ·Á´Â ±âÁ¾¹øÈ£
MOV       D00070 D00792	// º¯°æÇÏ·Á´Â ±âÁ¾¹øÈ£
RSET      0
MPOP
MUL       D00132 D00792 D02922
DADD      D02922 D00134 Z003
GMOV      R00000[Z003] D03100 D00132
MOVP      D00070 D00071	// º¯°æÇÏ·Á´Â ±âÁ¾¹øÈ£ / ÇöÀç DEV¹øÈ£
// output comment: 700°³ÀÇ µ¥ÀÌÅÍ¸¦ ºÒ·¯¿Ã °Å¸®¸¦ ±¸ÇÔ  =>Data ºÒ·¯¿Ã °÷ ÁÖ¼Ò±¸ÇÏ±â
// output comment: 6000 ¹øÁöºÎÅÍ µ¥ÀÌÅÍÀúÀå°ø°£ÀÌ´Ï±î ¾îµð¸¦ ºÒ·¯¿Í¾ßÇÏ´ÂÁö °è»ê
// output comment: µ¥ÀÌÅÍ ºÒ·¯¿À°í ³ª¼­ ¹øÈ£º¯°æ Àû¿ë
// Device  Copy
; L51
LOAD      M02199	// ±âÁ¾º¹»ç1p
DMOV      D19251 D00067	// ¿øº»
MPUSH
AND>      D00067 0	// ¿øº»
SUB       D00067 1 D00730	// ¿øº»
MLOAD
AND>      D00068 0	// Å¸°Ù
SUB       D00068 1 D00732	// Å¸°Ù
MPOP
AND<>     D00067 0	// ¿øº»
AND<>     D00068 0	// Å¸°Ù
AND<>     D00067 D00068	// ¿øº» / Å¸°Ù
AND<>     D00732 D00071	// ÇöÀç DEV¹øÈ£
OUTP      M0219B	// ±âÁ¾º¹»ç PLS
// output comment: BENDING±â¿¡¼­ ¹Þ¾Æ¿È
// output comment: È­¸é¿¡ Ç¥½ÃµÇ´Â µð¹ÙÀÌ½º ¹øÈ£°¡ 1¹øºÎÅÍÁö¸¸ ½ÇÁ¦·Î´Â 0 ¹øºÎÅÍ
// output comment: ¸Þ¸ð¸®¸¦ ÇÒ´çÇßÀ¸¹Ç·Î 1À» »©¼­ Ã³¸®

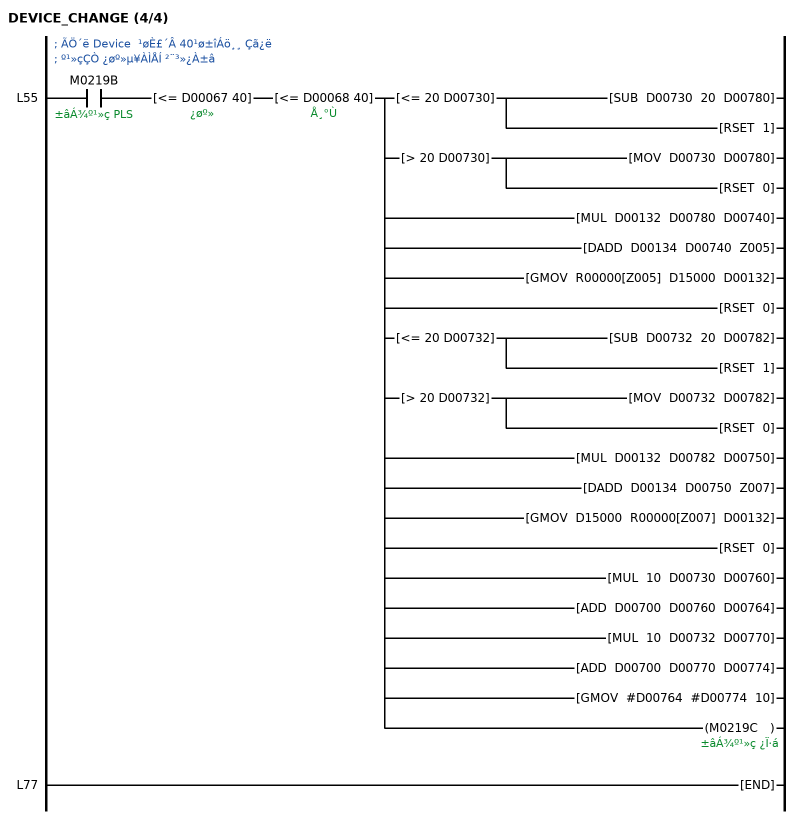
; L55
LOAD      M0219B	// ±âÁ¾º¹»ç PLS
AND<=     D00067 40	// ¿øº»
AND<=     D00068 40	// Å¸°Ù
MPUSH
AND<=     20 D00730
SUB       D00730 20 D00780
RSET      1
MLOAD
AND>      20 D00730
MOV       D00730 D00780
RSET      0
MLOAD
MUL       D00132 D00780 D00740
DADD      D00134 D00740 Z005
GMOV      R00000[Z005] D15000 D00132
RSET      0
AND<=     20 D00732
SUB       D00732 20 D00782
RSET      1
MLOAD
AND>      20 D00732
MOV       D00732 D00782
RSET      0
MPOP
MUL       D00132 D00782 D00750
DADD      D00134 D00750 Z007
GMOV      D15000 R00000[Z007] D00132
RSET      0
MUL       10 D00730 D00760
ADD       D00700 D00760 D00764
MUL       10 D00732 D00770
ADD       D00700 D00770 D00774
GMOV      #D00764 #D00774 10
OUT       M0219C	// ±âÁ¾º¹»ç ¿Ï·á
// output comment: ÃÖ´ë Device  ¹øÈ£´Â 40¹ø±îÁö¸¸ Çã¿ë
// output comment: º¹»çÇÒ ¿øº»µ¥ÀÌÅÍ ²¨³»¿À±â
; L77
END

PROGRAM SERVO (task: ½ºÄµ ÇÁ·Î±×·¥)

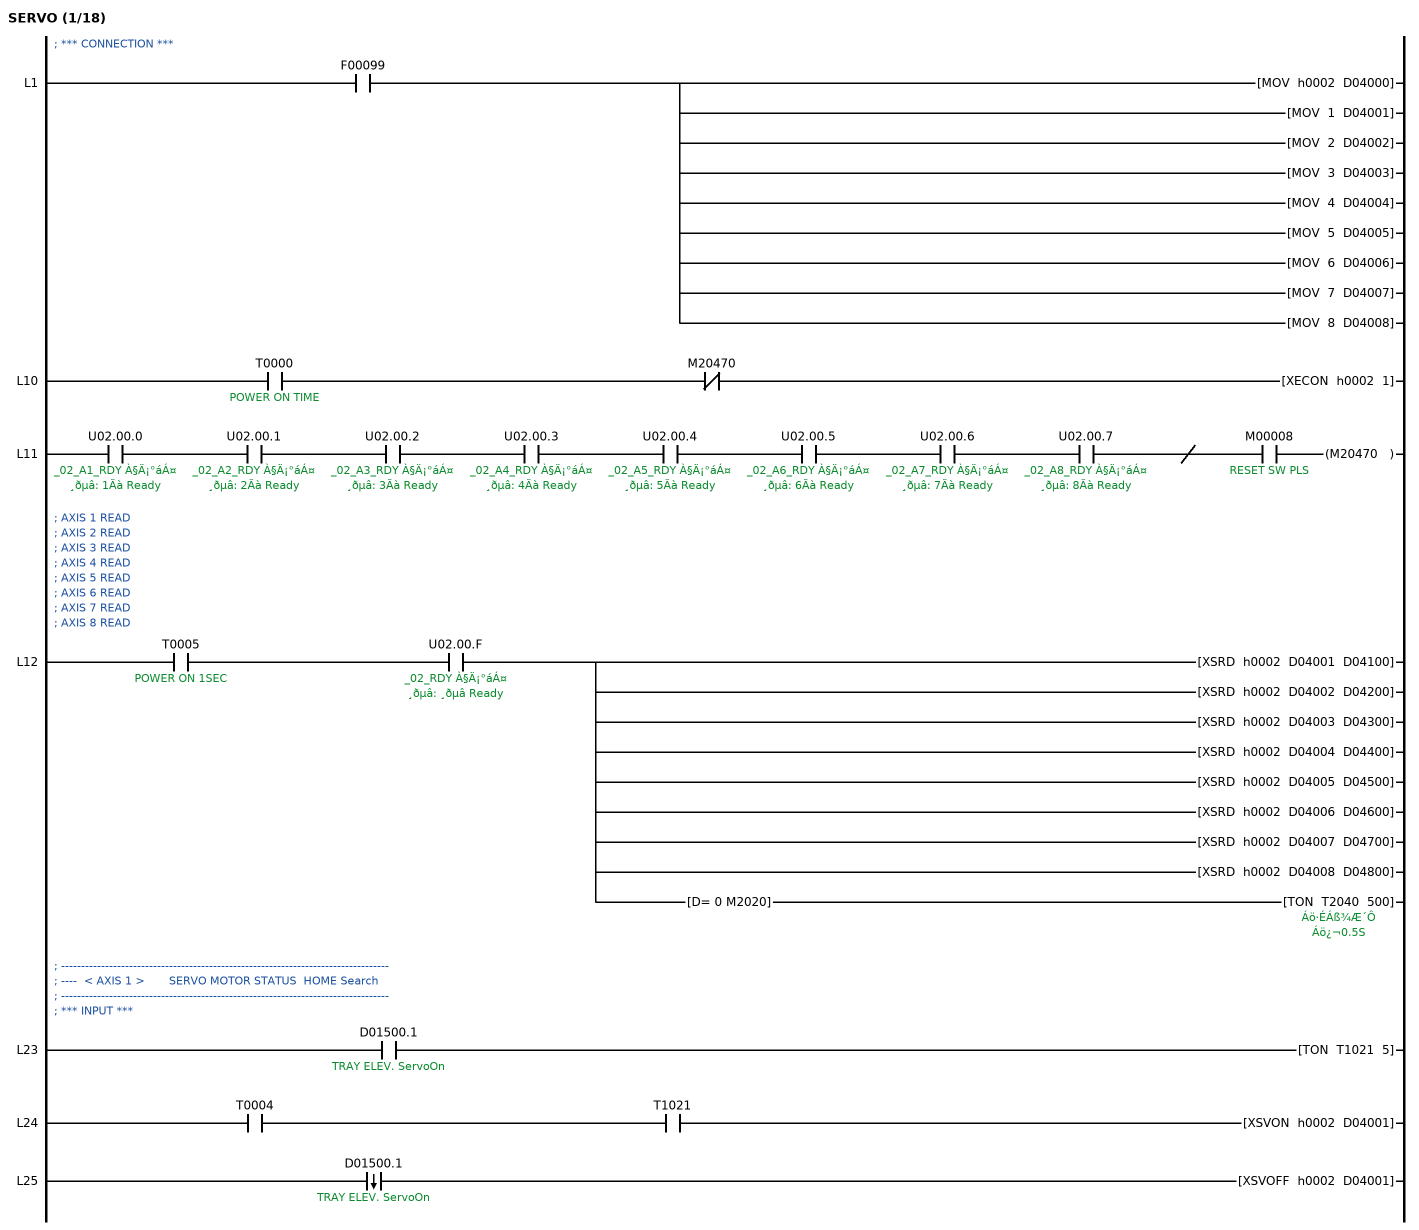
// *** CONNECTION ***
; L1
LOAD      F00099
MOV       h0002 D04000
MOV       1 D04001
MOV       2 D04002
MOV       3 D04003
MOV       4 D04004
MOV       5 D04005
MOV       6 D04006
MOV       7 D04007
MOV       8 D04008
; L10
LOAD      T0000	// POWER ON TIME
AND NOT   M20470
XECON     h0002 1
; L11
LOAD      U02.00.0	// _02_A1_RDY À§Ä¡°áÁ¤ ¸ðµâ: 1Ãà Ready
AND       U02.00.1	// _02_A2_RDY À§Ä¡°áÁ¤ ¸ðµâ: 2Ãà Ready
AND       U02.00.2	// _02_A3_RDY À§Ä¡°áÁ¤ ¸ðµâ: 3Ãà Ready
AND       U02.00.3	// _02_A4_RDY À§Ä¡°áÁ¤ ¸ðµâ: 4Ãà Ready
AND       U02.00.4	// _02_A5_RDY À§Ä¡°áÁ¤ ¸ðµâ: 5Ãà Ready
AND       U02.00.5	// _02_A6_RDY À§Ä¡°áÁ¤ ¸ðµâ: 6Ãà Ready
AND       U02.00.6	// _02_A7_RDY À§Ä¡°áÁ¤ ¸ðµâ: 7Ãà Ready
AND       U02.00.7	// _02_A8_RDY À§Ä¡°áÁ¤ ¸ðµâ: 8Ãà Ready
NOT
AND       M00008	// RESET SW PLS
OUT       M20470
; L12
LOAD      T0005	// POWER ON 1SEC
AND       U02.00.F	// _02_RDY À§Ä¡°áÁ¤ ¸ðµâ: ¸ðµâ Ready
XSRD      h0002 D04001 D04100
XSRD      h0002 D04002 D04200
XSRD      h0002 D04003 D04300
XSRD      h0002 D04004 D04400
XSRD      h0002 D04005 D04500
XSRD      h0002 D04006 D04600
XSRD      h0002 D04007 D04700
XSRD      h0002 D04008 D04800
ANDD=     0 M2020
TON       T2040 500	// Áö·ÉÁß¾Æ´Ô Áö¿¬0.5S
// output comment: AXIS 1 READ
// output comment: AXIS 2 READ
// output comment: AXIS 3 READ
// output comment: AXIS 4 READ
// output comment: AXIS 5 READ
// output comment: AXIS 6 READ
// output comment: AXIS 7 READ
// output comment: AXIS 8 READ
// ----------------------------------------------------------------------------------
// 
// ----  < AXIS 1 >       SERVO MOTOR STATUS  HOME Search
// 
// ----------------------------------------------------------------------------------
// *** INPUT ***
; L23
LOAD      D01500.1	// TRAY ELEV. ServoOn
TON       T1021 5
; L24
LOAD      T0004
AND       T1021
XSVON     h0002 D04001
; L25
LOADN     D01500.1	// TRAY ELEV. ServoOn
XSVOFF    h0002 D04001

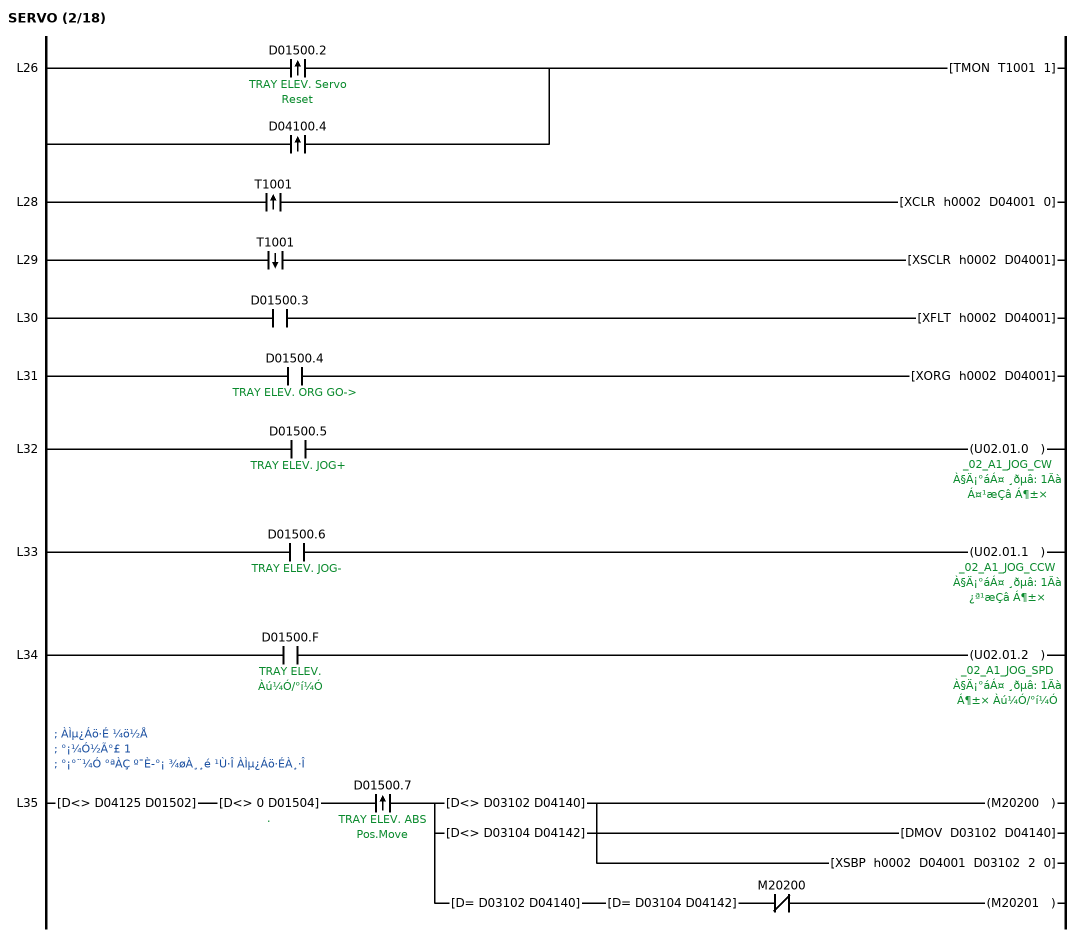
; L26
LOADP     D01500.2	// TRAY ELEV. Servo Reset
ORP       D04100.4
TMON      T1001 1
; L28
LOADP     T1001
XCLR      h0002 D04001 0
; L29
LOADN     T1001
XSCLR     h0002 D04001
; L30
LOAD      D01500.3
XFLT      h0002 D04001
; L31
LOAD      D01500.4	// TRAY ELEV. ORG GO->
XORG      h0002 D04001
; L32
LOAD      D01500.5	// TRAY ELEV. JOG+
OUT       U02.01.0	// _02_A1_JOG_CW À§Ä¡°áÁ¤ ¸ðµâ: 1Ãà Á¤¹æÇâ Á¶±×
; L33
LOAD      D01500.6	// TRAY ELEV. JOG-
OUT       U02.01.1	// _02_A1_JOG_CCW À§Ä¡°áÁ¤ ¸ðµâ: 1Ãà ¿ª¹æÇâ Á¶±×
; L34
LOAD      D01500.F	// TRAY ELEV. Àú¼Ó/°í¼Ó
OUT       U02.01.2	// _02_A1_JOG_SPD À§Ä¡°áÁ¤ ¸ðµâ: 1Ãà Á¶±× Àú¼Ó/°í¼Ó
; L35
LOADD<>   D04125 D01502
ANDD<>    0 D01504	// .
ANDP      D01500.7	// TRAY ELEV. ABS Pos.Move
MPUSH
LOADD<>   D03102 D04140
ORD<>     D03104 D04142
AND LOAD
OUT       M20200
DMOV      D03102 D04140
XSBP      h0002 D04001 D03102 2 0
MPOP
ANDD=     D03102 D04140
ANDD=     D03104 D04142
AND NOT   M20200
OUT       M20201
// output comment: ÀÌµ¿Áö·É ¼ö½Å
// output comment: °¡¼Ó½Ã°£ 1
// output comment: °¡°¨¼Ó °ªÀÇ º¯È­°¡ ¾øÀ¸¸é ¹Ù·Î ÀÌµ¿Áö·ÉÀ¸·Î

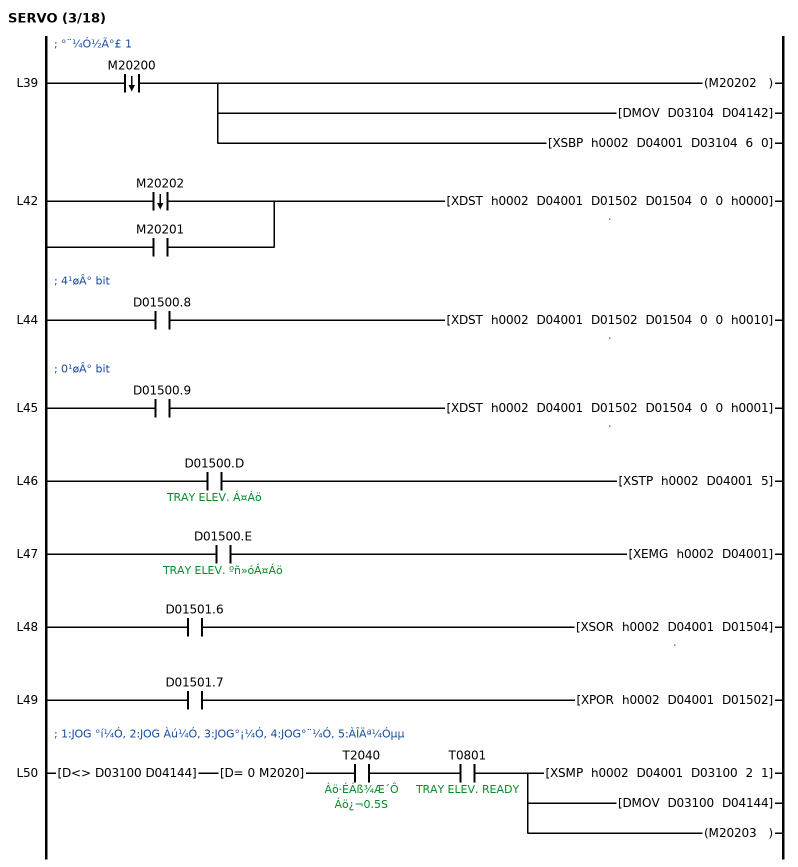
; L39
LOADN     M20200
OUT       M20202
DMOV      D03104 D04142
XSBP      h0002 D04001 D03104 6 0
// output comment: °¨¼Ó½Ã°£ 1
; L42
LOADN     M20202
OR        M20201
XDST      h0002 D04001 D01502 D01504 0 0 h0000	// .
; L44
LOAD      D01500.8
XDST      h0002 D04001 D01502 D01504 0 0 h0010	// .
// output comment: 4¹øÂ° bit
; L45
LOAD      D01500.9
XDST      h0002 D04001 D01502 D01504 0 0 h0001	// .
// output comment: 0¹øÂ° bit
; L46
LOAD      D01500.D	// TRAY ELEV. Á¤Áö
XSTP      h0002 D04001 5
; L47
LOAD      D01500.E	// TRAY ELEV. ºñ»óÁ¤Áö
XEMG      h0002 D04001
; L48
LOAD      D01501.6
XSOR      h0002 D04001 D01504	// .
; L49
LOAD      D01501.7
XPOR      h0002 D04001 D01502
; L50
LOADD<>   D03100 D04144
ANDD=     0 M2020
AND       T2040	// Áö·ÉÁß¾Æ´Ô Áö¿¬0.5S
AND       T0801	// TRAY ELEV. READY
XSMP      h0002 D04001 D03100 2 1
DMOV      D03100 D04144
OUT       M20203
// output comment: 1:JOG °í¼Ó, 2:JOG Àú¼Ó, 3:JOG°¡¼Ó, 4:JOG°¨¼Ó, 5:ÀÎÄª¼Óµµ

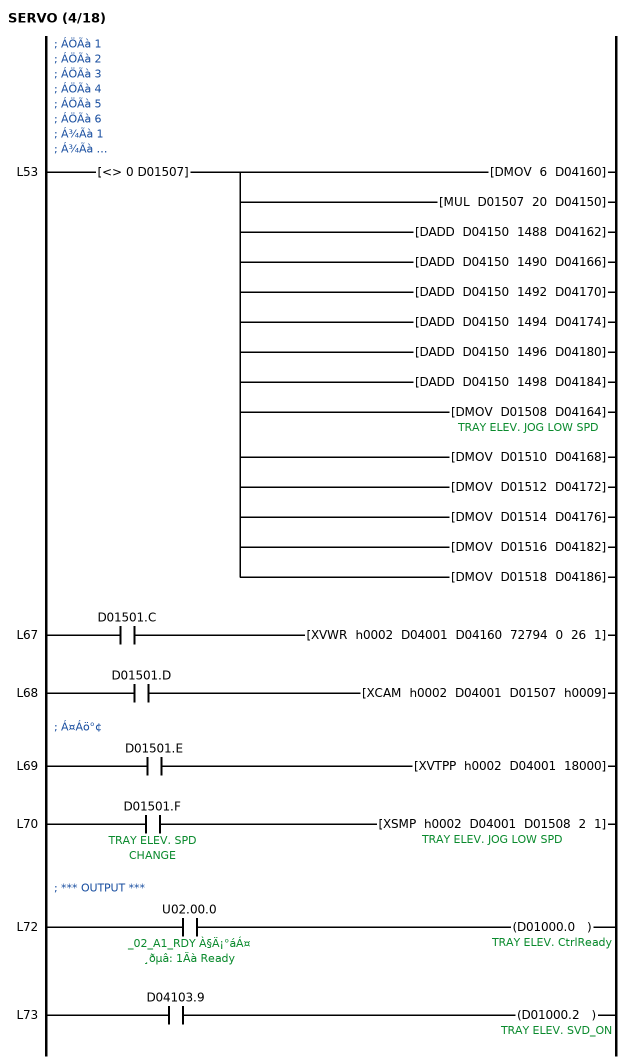
; L53
LOAD<>    0 D01507
DMOV      6 D04160
MUL       D01507 20 D04150
DADD      D04150 1488 D04162
DADD      D04150 1490 D04166
DADD      D04150 1492 D04170
DADD      D04150 1494 D04174
DADD      D04150 1496 D04180
DADD      D04150 1498 D04184
DMOV      D01508 D04164	// TRAY ELEV. JOG LOW SPD
DMOV      D01510 D04168
DMOV      D01512 D04172
DMOV      D01514 D04176
DMOV      D01516 D04182
DMOV      D01518 D04186
// output comment: ÁÖÃà 1
// output comment: ÁÖÃà 2
// output comment: ÁÖÃà 3
// output comment: ÁÖÃà 4
// output comment: ÁÖÃà 5
// output comment: ÁÖÃà 6
// output comment: Á¾Ãà 1
// output comment: Á¾Ãà 2
// output comment: Á¾Ãà 3
// output comment: Á¾Ãà 4
// output comment: Á¾Ãà 5
// output comment: Á¾Ãà 6
; L67
LOAD      D01501.C
XVWR      h0002 D04001 D04160 72794 0 26 1
; L68
LOAD      D01501.D
XCAM      h0002 D04001 D01507 h0009
; L69
LOAD      D01501.E
XVTPP     h0002 D04001 18000
// output comment: Á¤Áö°¢
; L70
LOAD      D01501.F	// TRAY ELEV. SPD CHANGE
XSMP      h0002 D04001 D01508 2 1	// TRAY ELEV. JOG LOW SPD
// *** OUTPUT ***
; L72
LOAD      U02.00.0	// _02_A1_RDY À§Ä¡°áÁ¤ ¸ðµâ: 1Ãà Ready
OUT       D01000.0	// TRAY ELEV. CtrlReady
; L73
LOAD      D04103.9
OUT       D01000.2	// TRAY ELEV. SVD_ON

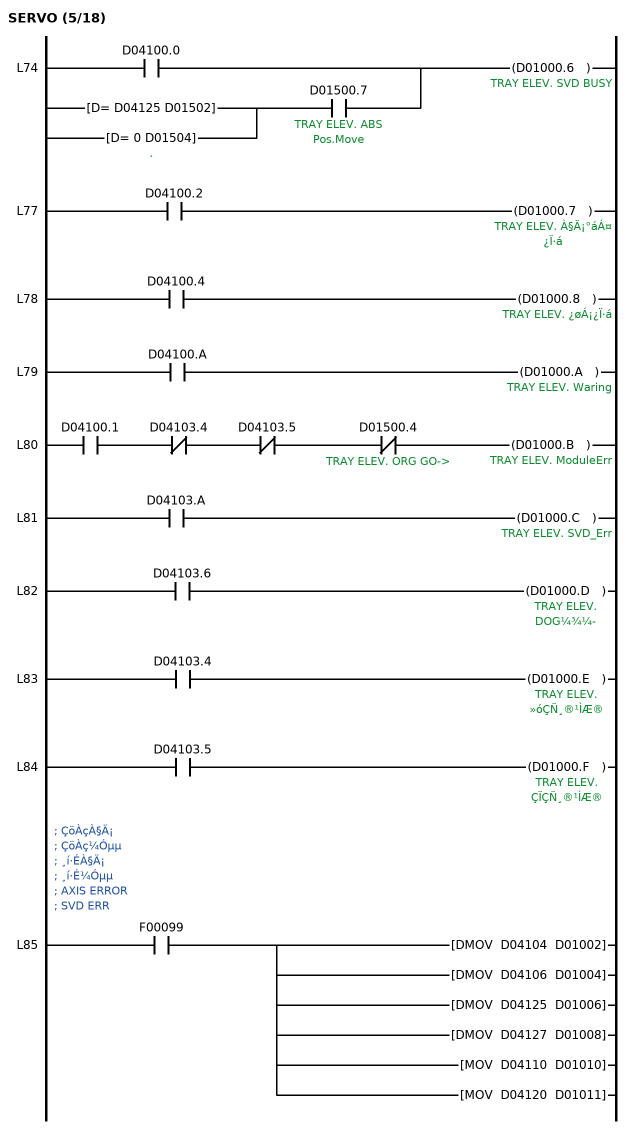
; L74
LOAD      D04100.0
LOADD=    D04125 D01502
ORD=      0 D01504	// .
AND       D01500.7	// TRAY ELEV. ABS Pos.Move
OR LOAD
OUT       D01000.6	// TRAY ELEV. SVD BUSY
; L77
LOAD      D04100.2
OUT       D01000.7	// TRAY ELEV. À§Ä¡°áÁ¤ ¿Ï·á
; L78
LOAD      D04100.4
OUT       D01000.8	// TRAY ELEV. ¿øÁ¡¿Ï·á
; L79
LOAD      D04100.A
OUT       D01000.A	// TRAY ELEV. Waring
; L80
LOAD      D04100.1
AND NOT   D04103.4
AND NOT   D04103.5
AND NOT   D01500.4	// TRAY ELEV. ORG GO->
OUT       D01000.B	// TRAY ELEV. ModuleErr
; L81
LOAD      D04103.A
OUT       D01000.C	// TRAY ELEV. SVD_Err
; L82
LOAD      D04103.6
OUT       D01000.D	// TRAY ELEV. DOG¼¾¼­
; L83
LOAD      D04103.4
OUT       D01000.E	// TRAY ELEV. »óÇÑ¸®¹ÌÆ®
; L84
LOAD      D04103.5
OUT       D01000.F	// TRAY ELEV. ÇÏÇÑ¸®¹ÌÆ®
; L85
LOAD      F00099
DMOV      D04104 D01002
DMOV      D04106 D01004
DMOV      D04125 D01006
DMOV      D04127 D01008
MOV       D04110 D01010
MOV       D04120 D01011
// output comment: ÇöÀçÀ§Ä¡
// output comment: ÇöÀç¼Óµµ
// output comment: ¸í·ÉÀ§Ä¡
// output comment: ¸í·É¼Óµµ
// output comment: AXIS ERROR
// output comment: SVD ERR

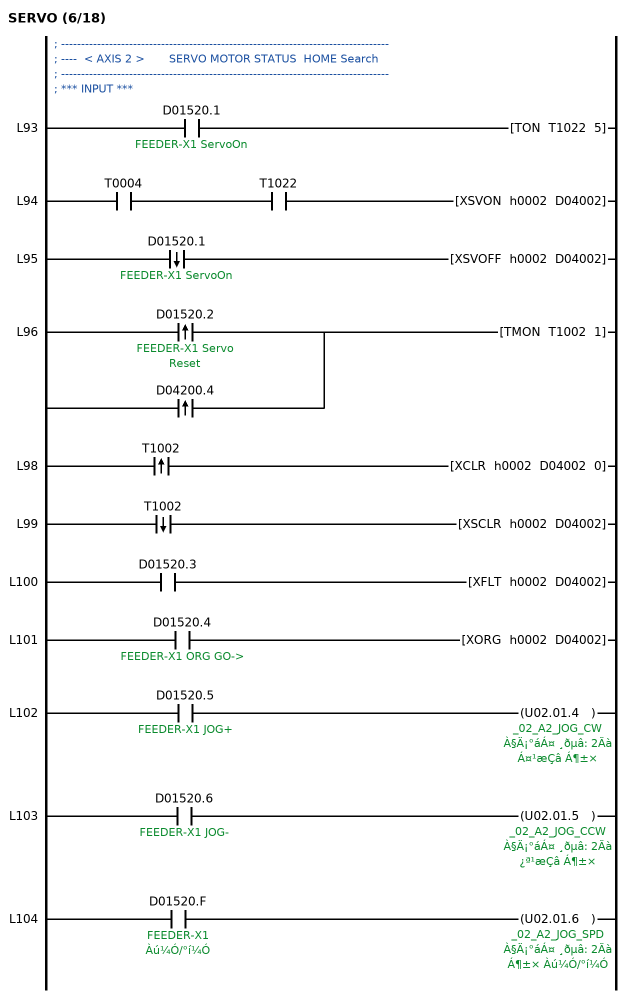
// ----------------------------------------------------------------------------------
// 
// ----  < AXIS 2 >       SERVO MOTOR STATUS  HOME Search
// 
// ----------------------------------------------------------------------------------
// *** INPUT ***
; L93
LOAD      D01520.1	// FEEDER-X1 ServoOn
TON       T1022 5
; L94
LOAD      T0004
AND       T1022
XSVON     h0002 D04002
; L95
LOADN     D01520.1	// FEEDER-X1 ServoOn
XSVOFF    h0002 D04002
; L96
LOADP     D01520.2	// FEEDER-X1 Servo Reset
ORP       D04200.4
TMON      T1002 1
; L98
LOADP     T1002
XCLR      h0002 D04002 0
; L99
LOADN     T1002
XSCLR     h0002 D04002
; L100
LOAD      D01520.3
XFLT      h0002 D04002
; L101
LOAD      D01520.4	// FEEDER-X1 ORG GO->
XORG      h0002 D04002
; L102
LOAD      D01520.5	// FEEDER-X1 JOG+
OUT       U02.01.4	// _02_A2_JOG_CW À§Ä¡°áÁ¤ ¸ðµâ: 2Ãà Á¤¹æÇâ Á¶±×
; L103
LOAD      D01520.6	// FEEDER-X1 JOG-
OUT       U02.01.5	// _02_A2_JOG_CCW À§Ä¡°áÁ¤ ¸ðµâ: 2Ãà ¿ª¹æÇâ Á¶±×
; L104
LOAD      D01520.F	// FEEDER-X1 Àú¼Ó/°í¼Ó
OUT       U02.01.6	// _02_A2_JOG_SPD À§Ä¡°áÁ¤ ¸ðµâ: 2Ãà Á¶±× Àú¼Ó/°í¼Ó

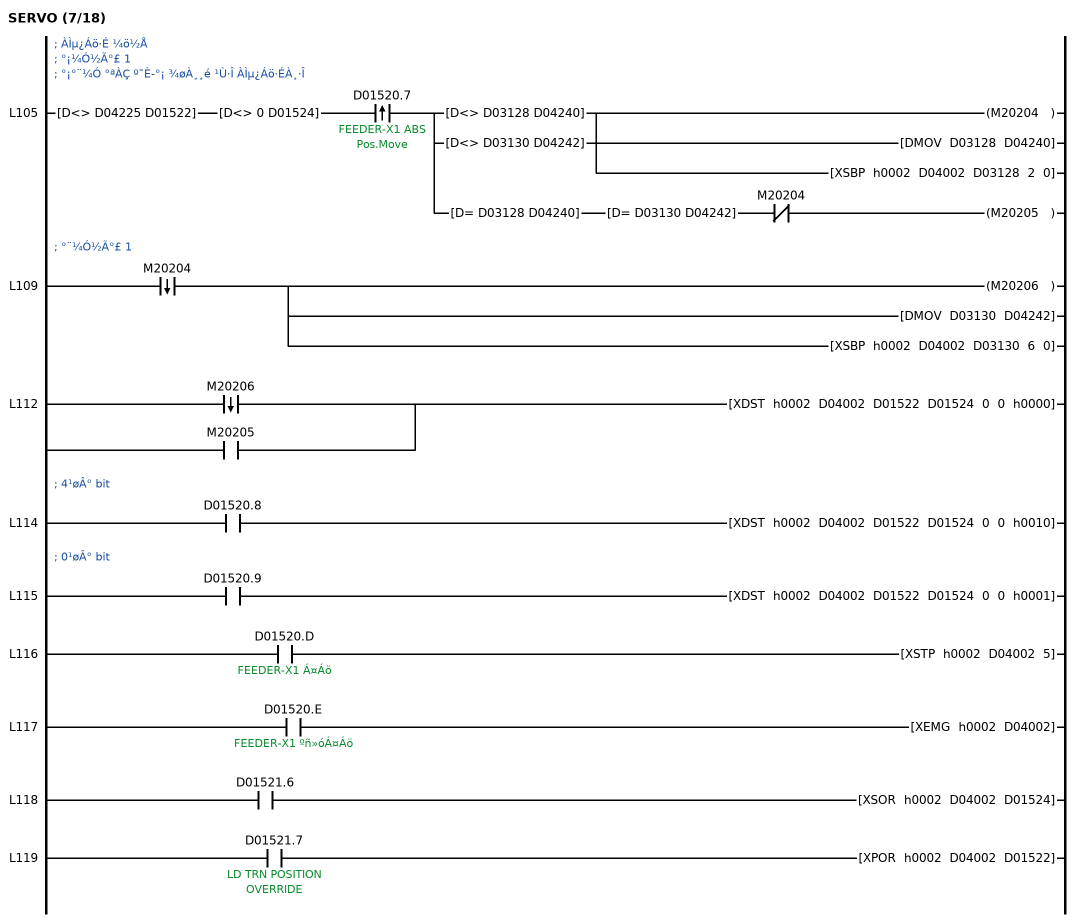
; L105
LOADD<>   D04225 D01522
ANDD<>    0 D01524
ANDP      D01520.7	// FEEDER-X1 ABS Pos.Move
MPUSH
LOADD<>   D03128 D04240
ORD<>     D03130 D04242
AND LOAD
OUT       M20204
DMOV      D03128 D04240
XSBP      h0002 D04002 D03128 2 0
MPOP
ANDD=     D03128 D04240
ANDD=     D03130 D04242
AND NOT   M20204
OUT       M20205
// output comment: ÀÌµ¿Áö·É ¼ö½Å
// output comment: °¡¼Ó½Ã°£ 1
// output comment: °¡°¨¼Ó °ªÀÇ º¯È­°¡ ¾øÀ¸¸é ¹Ù·Î ÀÌµ¿Áö·ÉÀ¸·Î
; L109
LOADN     M20204
OUT       M20206
DMOV      D03130 D04242
XSBP      h0002 D04002 D03130 6 0
// output comment: °¨¼Ó½Ã°£ 1
; L112
LOADN     M20206
OR        M20205
XDST      h0002 D04002 D01522 D01524 0 0 h0000
; L114
LOAD      D01520.8
XDST      h0002 D04002 D01522 D01524 0 0 h0010
// output comment: 4¹øÂ° bit
; L115
LOAD      D01520.9
XDST      h0002 D04002 D01522 D01524 0 0 h0001
// output comment: 0¹øÂ° bit
; L116
LOAD      D01520.D	// FEEDER-X1 Á¤Áö
XSTP      h0002 D04002 5
; L117
LOAD      D01520.E	// FEEDER-X1 ºñ»óÁ¤Áö
XEMG      h0002 D04002
; L118
LOAD      D01521.6
XSOR      h0002 D04002 D01524
; L119
LOAD      D01521.7	// LD TRN POSITION OVERRIDE
XPOR      h0002 D04002 D01522

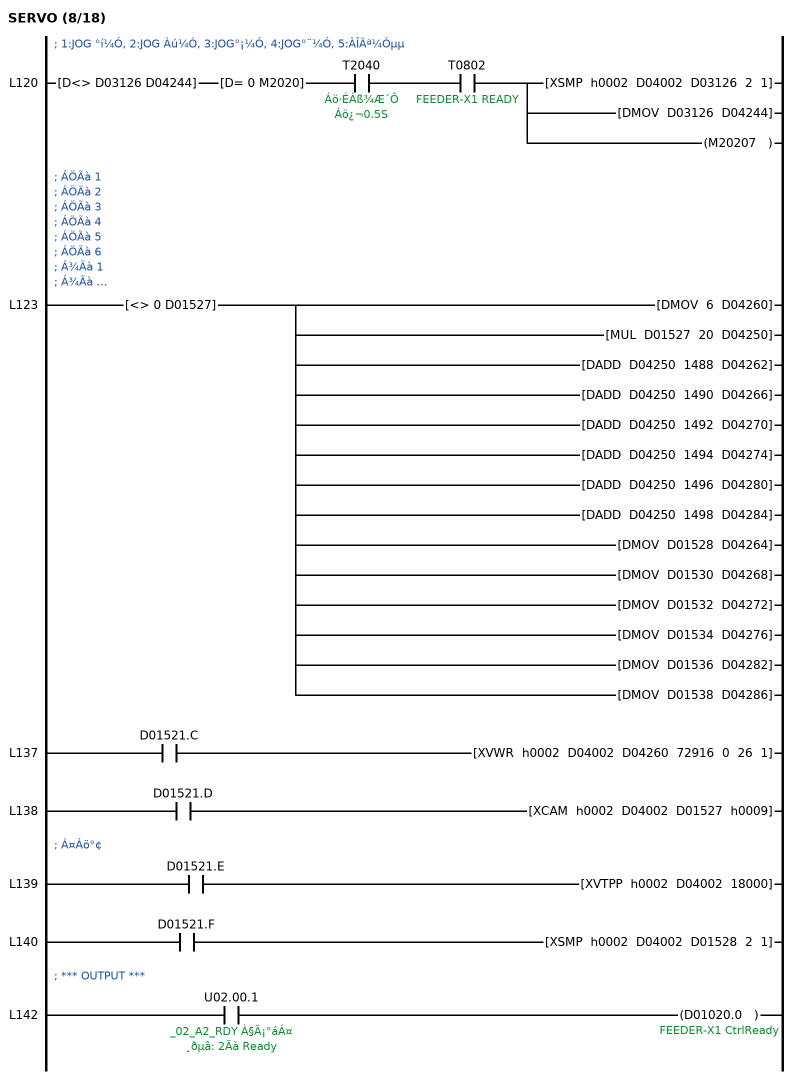
; L120
LOADD<>   D03126 D04244
ANDD=     0 M2020
AND       T2040	// Áö·ÉÁß¾Æ´Ô Áö¿¬0.5S
AND       T0802	// FEEDER-X1 READY
XSMP      h0002 D04002 D03126 2 1
DMOV      D03126 D04244
OUT       M20207
// output comment: 1:JOG °í¼Ó, 2:JOG Àú¼Ó, 3:JOG°¡¼Ó, 4:JOG°¨¼Ó, 5:ÀÎÄª¼Óµµ
; L123
LOAD<>    0 D01527
DMOV      6 D04260
MUL       D01527 20 D04250
DADD      D04250 1488 D04262
DADD      D04250 1490 D04266
DADD      D04250 1492 D04270
DADD      D04250 1494 D04274
DADD      D04250 1496 D04280
DADD      D04250 1498 D04284
DMOV      D01528 D04264
DMOV      D01530 D04268
DMOV      D01532 D04272
DMOV      D01534 D04276
DMOV      D01536 D04282
DMOV      D01538 D04286
// output comment: ÁÖÃà 1
// output comment: ÁÖÃà 2
// output comment: ÁÖÃà 3
// output comment: ÁÖÃà 4
// output comment: ÁÖÃà 5
// output comment: ÁÖÃà 6
// output comment: Á¾Ãà 1
// output comment: Á¾Ãà 2
// output comment: Á¾Ãà 3
// output comment: Á¾Ãà 4
// output comment: Á¾Ãà 5
// output comment: Á¾Ãà 6
; L137
LOAD      D01521.C
XVWR      h0002 D04002 D04260 72916 0 26 1
; L138
LOAD      D01521.D
XCAM      h0002 D04002 D01527 h0009
; L139
LOAD      D01521.E
XVTPP     h0002 D04002 18000
// output comment: Á¤Áö°¢
; L140
LOAD      D01521.F
XSMP      h0002 D04002 D01528 2 1
// *** OUTPUT ***
; L142
LOAD      U02.00.1	// _02_A2_RDY À§Ä¡°áÁ¤ ¸ðµâ: 2Ãà Ready
OUT       D01020.0	// FEEDER-X1 CtrlReady

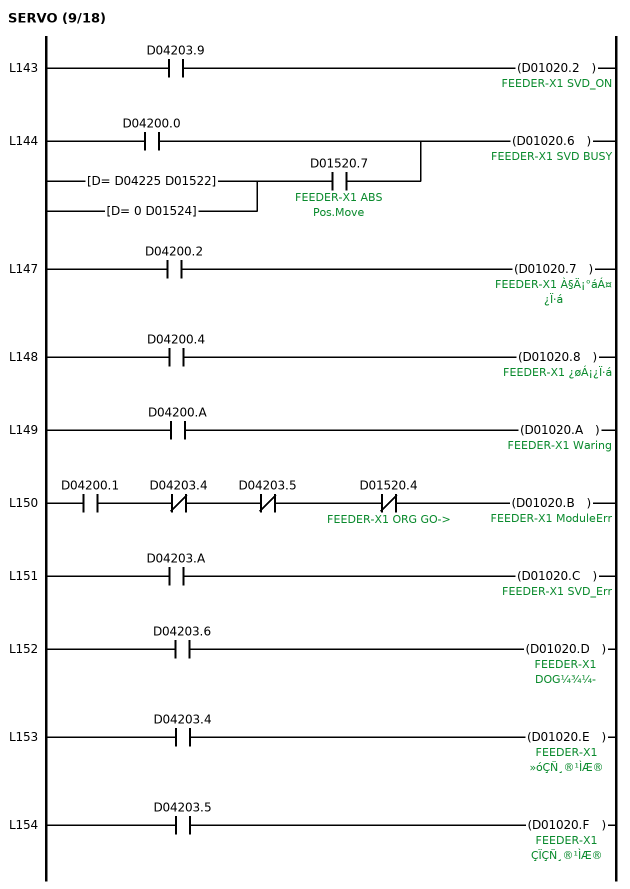
; L143
LOAD      D04203.9
OUT       D01020.2	// FEEDER-X1 SVD_ON
; L144
LOAD      D04200.0
LOADD=    D04225 D01522
ORD=      0 D01524
AND       D01520.7	// FEEDER-X1 ABS Pos.Move
OR LOAD
OUT       D01020.6	// FEEDER-X1 SVD BUSY
; L147
LOAD      D04200.2
OUT       D01020.7	// FEEDER-X1 À§Ä¡°áÁ¤ ¿Ï·á
; L148
LOAD      D04200.4
OUT       D01020.8	// FEEDER-X1 ¿øÁ¡¿Ï·á
; L149
LOAD      D04200.A
OUT       D01020.A	// FEEDER-X1 Waring
; L150
LOAD      D04200.1
AND NOT   D04203.4
AND NOT   D04203.5
AND NOT   D01520.4	// FEEDER-X1 ORG GO->
OUT       D01020.B	// FEEDER-X1 ModuleErr
; L151
LOAD      D04203.A
OUT       D01020.C	// FEEDER-X1 SVD_Err
; L152
LOAD      D04203.6
OUT       D01020.D	// FEEDER-X1 DOG¼¾¼­
; L153
LOAD      D04203.4
OUT       D01020.E	// FEEDER-X1 »óÇÑ¸®¹ÌÆ®
; L154
LOAD      D04203.5
OUT       D01020.F	// FEEDER-X1 ÇÏÇÑ¸®¹ÌÆ®

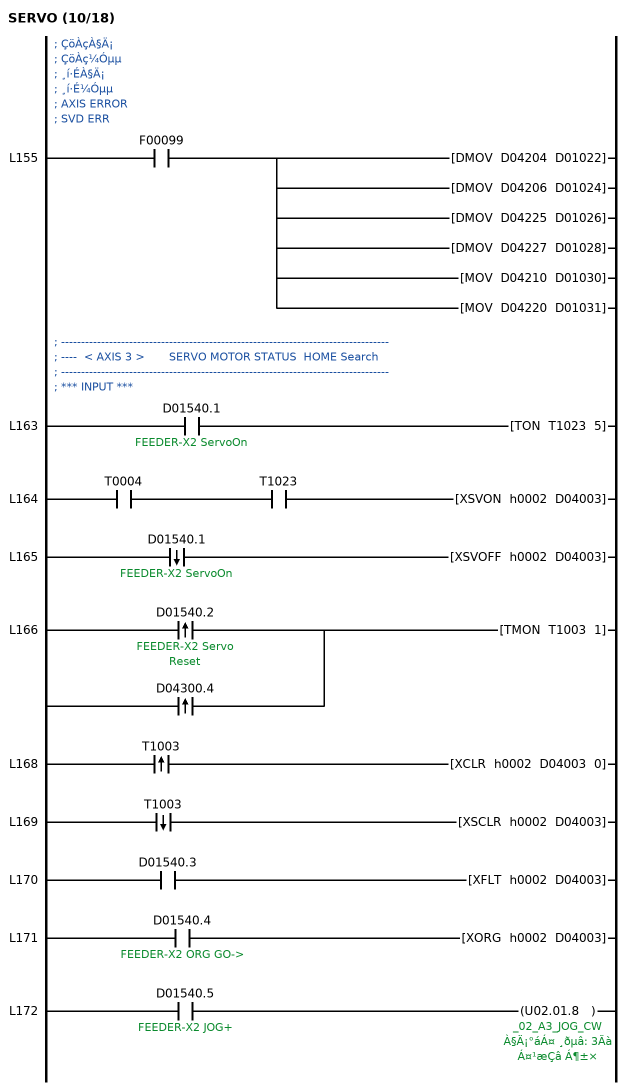
; L155
LOAD      F00099
DMOV      D04204 D01022
DMOV      D04206 D01024
DMOV      D04225 D01026
DMOV      D04227 D01028
MOV       D04210 D01030
MOV       D04220 D01031
// output comment: ÇöÀçÀ§Ä¡
// output comment: ÇöÀç¼Óµµ
// output comment: ¸í·ÉÀ§Ä¡
// output comment: ¸í·É¼Óµµ
// output comment: AXIS ERROR
// output comment: SVD ERR
// ----------------------------------------------------------------------------------
// 
// ----  < AXIS 3 >       SERVO MOTOR STATUS  HOME Search
// 
// ----------------------------------------------------------------------------------
// *** INPUT ***
; L163
LOAD      D01540.1	// FEEDER-X2 ServoOn
TON       T1023 5
; L164
LOAD      T0004
AND       T1023
XSVON     h0002 D04003
; L165
LOADN     D01540.1	// FEEDER-X2 ServoOn
XSVOFF    h0002 D04003
; L166
LOADP     D01540.2	// FEEDER-X2 Servo Reset
ORP       D04300.4
TMON      T1003 1
; L168
LOADP     T1003
XCLR      h0002 D04003 0
; L169
LOADN     T1003
XSCLR     h0002 D04003
; L170
LOAD      D01540.3
XFLT      h0002 D04003
; L171
LOAD      D01540.4	// FEEDER-X2 ORG GO->
XORG      h0002 D04003
; L172
LOAD      D01540.5	// FEEDER-X2 JOG+
OUT       U02.01.8	// _02_A3_JOG_CW À§Ä¡°áÁ¤ ¸ðµâ: 3Ãà Á¤¹æÇâ Á¶±×

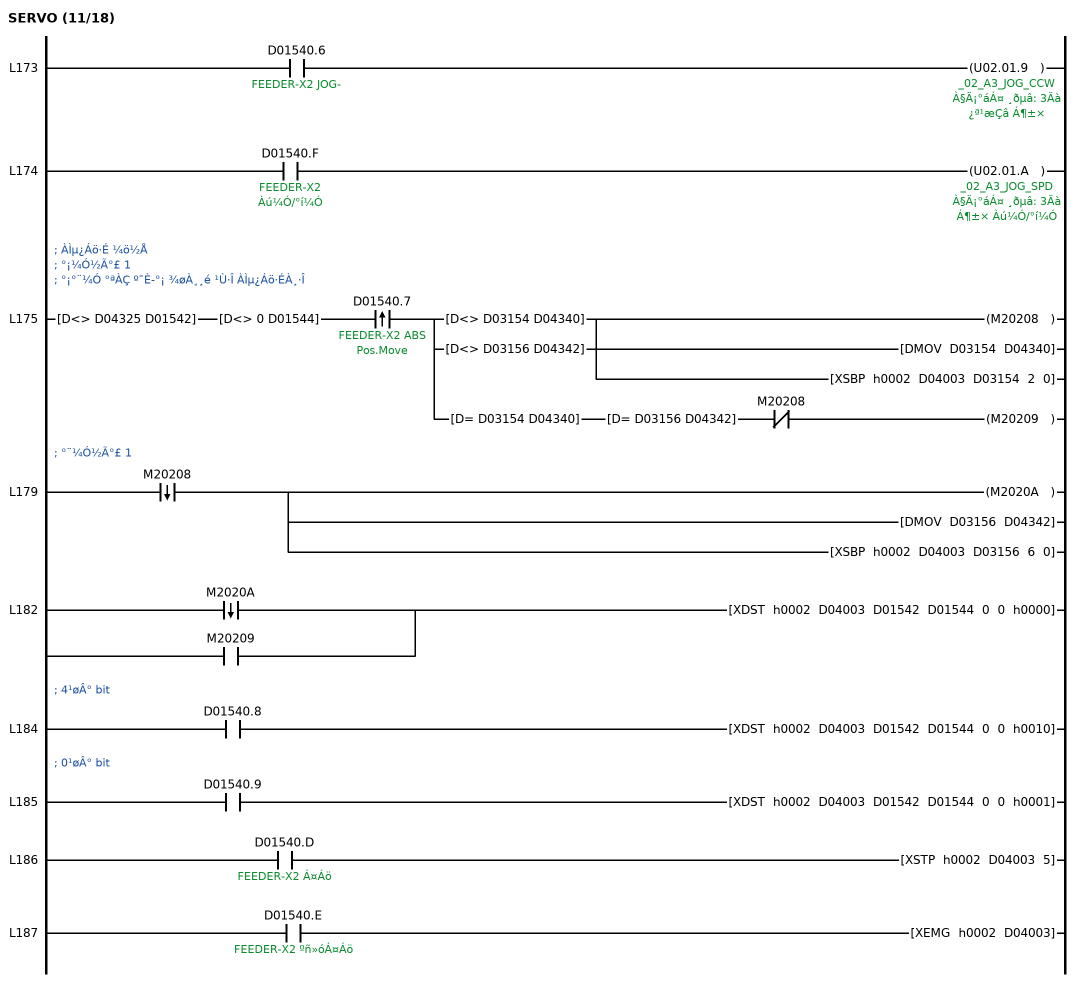
; L173
LOAD      D01540.6	// FEEDER-X2 JOG-
OUT       U02.01.9	// _02_A3_JOG_CCW À§Ä¡°áÁ¤ ¸ðµâ: 3Ãà ¿ª¹æÇâ Á¶±×
; L174
LOAD      D01540.F	// FEEDER-X2 Àú¼Ó/°í¼Ó
OUT       U02.01.A	// _02_A3_JOG_SPD À§Ä¡°áÁ¤ ¸ðµâ: 3Ãà Á¶±× Àú¼Ó/°í¼Ó
; L175
LOADD<>   D04325 D01542
ANDD<>    0 D01544
ANDP      D01540.7	// FEEDER-X2 ABS Pos.Move
MPUSH
LOADD<>   D03154 D04340
ORD<>     D03156 D04342
AND LOAD
OUT       M20208
DMOV      D03154 D04340
XSBP      h0002 D04003 D03154 2 0
MPOP
ANDD=     D03154 D04340
ANDD=     D03156 D04342
AND NOT   M20208
OUT       M20209
// output comment: ÀÌµ¿Áö·É ¼ö½Å
// output comment: °¡¼Ó½Ã°£ 1
// output comment: °¡°¨¼Ó °ªÀÇ º¯È­°¡ ¾øÀ¸¸é ¹Ù·Î ÀÌµ¿Áö·ÉÀ¸·Î
; L179
LOADN     M20208
OUT       M2020A
DMOV      D03156 D04342
XSBP      h0002 D04003 D03156 6 0
// output comment: °¨¼Ó½Ã°£ 1
; L182
LOADN     M2020A
OR        M20209
XDST      h0002 D04003 D01542 D01544 0 0 h0000
; L184
LOAD      D01540.8
XDST      h0002 D04003 D01542 D01544 0 0 h0010
// output comment: 4¹øÂ° bit
; L185
LOAD      D01540.9
XDST      h0002 D04003 D01542 D01544 0 0 h0001
// output comment: 0¹øÂ° bit
; L186
LOAD      D01540.D	// FEEDER-X2 Á¤Áö
XSTP      h0002 D04003 5
; L187
LOAD      D01540.E	// FEEDER-X2 ºñ»óÁ¤Áö
XEMG      h0002 D04003

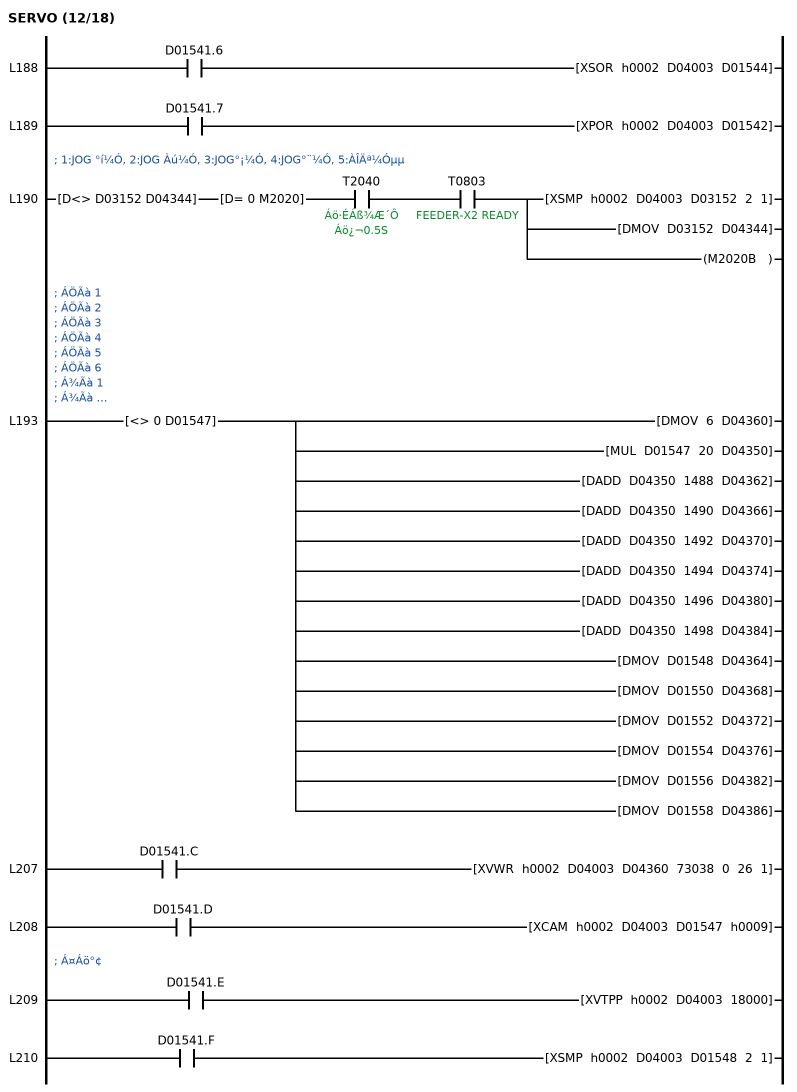
; L188
LOAD      D01541.6
XSOR      h0002 D04003 D01544
; L189
LOAD      D01541.7
XPOR      h0002 D04003 D01542
; L190
LOADD<>   D03152 D04344
ANDD=     0 M2020
AND       T2040	// Áö·ÉÁß¾Æ´Ô Áö¿¬0.5S
AND       T0803	// FEEDER-X2 READY
XSMP      h0002 D04003 D03152 2 1
DMOV      D03152 D04344
OUT       M2020B
// output comment: 1:JOG °í¼Ó, 2:JOG Àú¼Ó, 3:JOG°¡¼Ó, 4:JOG°¨¼Ó, 5:ÀÎÄª¼Óµµ
; L193
LOAD<>    0 D01547
DMOV      6 D04360
MUL       D01547 20 D04350
DADD      D04350 1488 D04362
DADD      D04350 1490 D04366
DADD      D04350 1492 D04370
DADD      D04350 1494 D04374
DADD      D04350 1496 D04380
DADD      D04350 1498 D04384
DMOV      D01548 D04364
DMOV      D01550 D04368
DMOV      D01552 D04372
DMOV      D01554 D04376
DMOV      D01556 D04382
DMOV      D01558 D04386
// output comment: ÁÖÃà 1
// output comment: ÁÖÃà 2
// output comment: ÁÖÃà 3
// output comment: ÁÖÃà 4
// output comment: ÁÖÃà 5
// output comment: ÁÖÃà 6
// output comment: Á¾Ãà 1
// output comment: Á¾Ãà 2
// output comment: Á¾Ãà 3
// output comment: Á¾Ãà 4
// output comment: Á¾Ãà 5
// output comment: Á¾Ãà 6
; L207
LOAD      D01541.C
XVWR      h0002 D04003 D04360 73038 0 26 1
; L208
LOAD      D01541.D
XCAM      h0002 D04003 D01547 h0009
; L209
LOAD      D01541.E
XVTPP     h0002 D04003 18000
// output comment: Á¤Áö°¢
; L210
LOAD      D01541.F
XSMP      h0002 D04003 D01548 2 1

